// TwinCAT 3 PLC project DMXV2PLC
// ProgramVersion: 3.1.4023.0
// libraries:
//   Tc2_Math, * (Beckhoff Automation GmbH)
//   Tc2_Standard, * (Beckhoff Automation GmbH)
//   Tc2_System, * (Beckhoff Automation GmbH)
//   Tc2_Utilities, * (Beckhoff Automation GmbH)
//   Tc3_Module, * (Beckhoff Automation GmbH)
//   VisuDialogs, * (System)
//   VisuSymbols, * (System)
//   Base Interfaces,newest,System
// project tree:
//   DUTs/ arr_rt.TcDUT, ENUM_BufferMgmt.TcDUT (not stored), ENUM_IQ_OpMode.TcDUT, ENUM_I_ValRange.TcDUT, ENUM_I_Waveform.TcDUT (not stored), ENUM_SeqSM.TcDUT (not stored), ST_CSV_Record.TcDUT (not stored), typDMXInOut.TcDUT, typDMXInput.TcDUT, typDMXOutput.TcDUT, typFBDInOut.TcDUT, typFBDInput.TcDUT (not stored), typFBDOutput.TcDUT, typ_FBInt_Debounce.TcDUT (not stored), typ_FBInt_DMX.TcDUT (not stored)
//   / GlobalTextList.TcGTLO, PlcTask.TcTTO, Visualization Manager.TcVMO (not stored)
//   GVLs/ gc.TcGVL, gFB.TcGVL (not stored), GVL.TcGVL (not stored), g_ast.TcGVL
//   POUs/ DMXShop.TcPOU, DMXTest.TcPOU, FBOscillator.TcPOU, FB_DMX.TcPOU, FB_InputDebounce.TcPOU, f_to_Period.TcPOU (not stored), InterfaceLink.TcPOU, MAIN.TcPOU, Map.TcPOU (not stored), MapClamp.TcPOU (not stored), P_ArgToConvExample.TcPOU (not stored), P_BinaryModeRead.TcPOU (not stored), P_BinaryModeWrite.TcPOU (not stored), P_StringToConvExample.TcPOU (not stored), P_TextModeRead.TcPOU, P_TextModeWrite.TcPOU, SclByteDMX.TcPOU, SclBytePNP.TcPOU (not stored)
//   VISUs/ Visualization.TcVIS

CONFIGURATION DMXV2PLC
    RESOURCE PLC ON TwinCAT3
        TASK PlcTask(INTERVAL := T#10ms, PRIORITY := 20);
        PROGRAM InterfaceLink WITH PlcTask : InterfaceLink;
        PROGRAM P_TextModeRead WITH PlcTask : P_TextModeRead;
        PROGRAM DMXShop WITH PlcTask : DMXShop;
    END_RESOURCE
END_CONFIGURATION

// ---- DUTs/arr_rt.TcDUT
TYPE ARR_RT	 :
STRUCT
	arrRcvdR_T	: ARRAY[0..gc.uiMaxNrDMXTestCh] OF R_TRIG;
	arrExpctdBool : ARRAY[0..gc.uiMaxNrDMXTestCh] OF BOOL;
END_STRUCT
END_TYPE

// ---- DUTs/ENUM_IQ_OpMode.TcDUT
{attribute 'qualified_only'}
{attribute 'strict'}
TYPE ENUM_IQ_OpMode :
(
	EN_Cycle		:= 0,
	EN_LatchOn		:= 1,
	EN_OneShot		:= 2
);
END_TYPE

// ---- DUTs/ENUM_I_ValRange.TcDUT
{attribute 'qualified_only'}
{attribute 'strict'}
TYPE ENUM_I_ValRange :
(
	EN_8Bit		:= 0,
	EN_16Bit	:= 1
);
END_TYPE

// ---- DUTs/typDMXInOut.TcDUT
TYPE typDMXInOut :
STRUCT
	fOffset				: REAL; // 0-100% mapped to 8-bit (by Map Function)
	fLevel				: REAL; // 0-100% mapped to 8-bit (by Map Function)
	usiBitDepth			: USINT; // 1-8
	xCmdOn				: BOOL;
	xCmdOff				: BOOL;
	fOutputIncrement	: REAL;
	fFnGenerValTempSin	: LREAL;
	fFnGenerValRtn		: LREAL;
	uiMaxChannelVal		: UINT;
	uiMinChannelVal		: UINT;
	byMaxChanVal		: BYTE;
	byMinChanVal		: BYTE;
END_STRUCT
END_TYPE

// ---- DUTs/typDMXInput.TcDUT
TYPE typDMXInput :
STRUCT
	ENWaveform		: ENUM_I_Waveform;
	ENValRange		: ENUM_I_ValRange;
	fDutyCycle		: REAL; // just for Square Wave;
	fFrequency		: REAL;  // Frequency of cycling, expressed in Hz
	fOffset			: REAL; // 0-100% mapped to 8-bit (by Map Function)
	fLevel			: REAL; // 0-100% mapped to 8-bit (by Map Function)
	usiBitDepth		: USINT; // 1-8
	fPhase			: REAL; // 0-100% mapped to 8-bit (by Map Function)
	fDelay			: REAL; // 0-100% mapped to 8-bit (by Map Function)
	usiDelayDiv		: USINT; // to Delay the step of the Delay Divisor; for example, '2' would delay every second pulse by the amount spec'd by fDelay
	usiInputConfig	: USINT; // BYTE Value specified in USINT [0-255]
	xCmdOn				: BOOL;
	xCmdOff				: BOOL;
	fOutputIncrement	: REAL;
	fFnGenerValTempSin	: LREAL;
	fFnGenerValRtn		: LREAL;
	uiMaxChannelVal		: UINT;
	uiMinChannelVal		: UINT;
	byMaxChanVal		: BYTE;
	byMinChanVal		: BYTE;
END_STRUCT
END_TYPE

// ---- DUTs/typDMXOutput.TcDUT
TYPE typDMXOutput :
STRUCT
	byStatValue			: BYTE;
	fFnGeneratorVal		: REAL;
END_STRUCT
END_TYPE

// ---- DUTs/typFBDInOut.TcDUT
TYPE typFBDInOut :
	STRUCT
		xTrig		: BOOL;
	END_STRUCT
END_TYPE

// ---- DUTs/typFBDOutput.TcDUT
TYPE typFBDOutput :
STRUCT
	xGate	: BOOL;
END_STRUCT
END_TYPE

// ---- GVLs/gc.TcGVL
{attribute 'qualified_only'}
VAR_GLOBAL CONSTANT
	uiMaxNrOfDMXChannel				: UINT := 511;
	wChannelLength			AT %Q*	: WORD := 512;
	fPi								: REAL	:= 3.141592653589793238462643383279;
	uiMinNrDMXTestCh				: UINT	:= 0;
	uiMaxNrDMXTestCh				: UINT	:= 79; // Dictated by hardware constraints (80 channels input)
	uiChannelsUT	 				: UINT	:= 80;		(*Channels Under Test *)
	uiVisualizationIndexLim			: UINT	:= 7;
	uiDUTConfigCountSplit			: UINT	:= 255;
	uiChannelSplitCount				: UINT	:= 256;
	
	// DMXShop 
	RED		: USINT := 0;
	GREEN 	: USINT := 1;
	BLUE	: USINT := 2;
	WHITE	: USINT := 3;

END_VAR

// ---- GVLs/g_ast.TcGVL
{attribute 'qualified_only'}
VAR_GLOBAL
		// INPUT array structs for mapping to Physical I/O (PIO)
//	gast_SensorInput		AT %I* : ARRAY[0..gc.usiMaxNrOfSensor] OF typ_FBInt_Debounce;
	
	//2 Sensors on each valve (assumed)
//	gast_ValveSensorInput	AT %I* : ARRAY[0..(2*gc.usiMaxNrOfValveCtrl)] OF typ_FBInt_Debounce;
//	gast_AnalogInput		AT %I* : ARRAY[0..gc.usiMaxNrOfAnalogIn] OF typ_FBInt_Analog;
	
// OUTPUT array structs for mapping to Physical I/O (PIO)
//	gast_ValveCtrlOutput	AT %Q* : ARRAY[0..gc.usiMaxNrOfValveCtrl] OF typ_FBInt_ValveCtrl;
//	gast_DigCtrlOutput		AT %Q* : ARRAY[0..gc.usiMaxNrOfDigCtrl] OF typ_FBInt_DigCtrl;
	DMX						: ARRAY[0..gc.uiMaxNrOfDMXChannel] OF typ_FBInt_DMX;
	DMXPhysOut				: ARRAY[0..gc.uiMaxNrOfDMXChannel] OF BYTE; (* software buffer *)
	DMXHWOut		AT %Q*	: ARRAY[0..gc.uiMaxNrOfDMXChannel] OF BYTE; (* Defined to allow Multi-Link of I/O in Physical I/O tree *)
	arrFBIntPNP				: ARRAY[0..gc.uiMaxNrDMXTestCh] OF typ_FBInt_Debounce;
	arrFBIntNPN				: ARRAY[0..gc.uiMaxNrDMXTestCh] OF typ_FBInt_Debounce;
	arrInputPNP		AT %I*	: ARRAY[0..gc.uiMaxNrDMXTestCh] OF BOOL;
	arrInputNPN		AT %I*	: ARRAY[0..gc.uiMaxNrDMXTestCh] OF BOOL;
END_VAR

// ---- POUs/InterfaceLink.TcPOU
PROGRAM InterfaceLink
VAR
	iResult					: INT;
	iLoopFBAnalogIn			: INT;
	iLoopFBSensor			: INT;
	iLoopFBValveSensor		: INT;
	iLoopFBDigCtrl			: INT;
	iLoopFBValveCtrl		: INT;
	uiLoopDMXCtrlI			: UINT;
	uiLoopDMXCtrlII			: UINT;
	uiLoopDebouncePNPI		: UINT;
	uiLoopDebounceNPNI		: UINT;
	uiForLoopDMXI10			: UINT;
	uiForLoopDMXI11			: UINT;
	uiForLoopDMXI12			: UINT;
	uiForLoopDebouncePNP	: UINT;
	uiForLoopDebounceNPN	: UINT;
END_VAR

//Call all the I/O Function Blocks continuously; link to array-structs with every call;
(*
FOR iLoopFBAnalogIn := 0 TO gc.usiMaxNrOfAnalogIn BY 1 DO
	gFB.arrFB_AnalogInput[iLoopFBAnalogIn](I:=gast_AnalogInput[iLoopFBAnalogIn].I, IQ:=gast_AnalogInput[iLoopFBAnalogIn].IQ, Q=>gast_AnalogInput[iLoopFBAnalogIn].Q);
END_FOR

FOR iLoopFBSensor := 0 TO gc.usiMaxNrOfSensor BY 1 DO
	gFB.arrFB_Sensor[iLoopFBSensor](I:=gast_SensorInput[iLoopFBSensor].I, IQ:=gast_SensorInput[iLoopFBSensor].IQ, Q=>gast_SensorInput[iLoopFBSensor].Q);
END_FOR

FOR iLoopFBValveSensor := 0 TO (2*gc.usiMaxNrOfValveCtrl) BY 1 DO
	gFB.arrFB_Sensor[iLoopFBValveSensor](I:=gast_ValveSensorInput[iLoopFBValveSensor].I, IQ:=gast_ValveSensorInput[iLoopFBValveSensor].IQ, Q=>gast_ValveSensorInput[iLoopFBValveSensor].Q);
END_FOR

FOR iLoopFBDigCtrl := 0 TO gc.usiMaxNrOfSensor BY 1 DO
	gFB.arrFB_DigCtrl[iLoopFBDigCtrl](I:=gast_DigCtrlOutput[iLoopFBDigCtrl].I, IQ:=gast_DigCtrlOutput[iLoopFBDigCtrl].IQ, Q=>gast_DigCtrlOutput[iLoopFBDigCtrl].Q);
END_FOR

FOR iLoopFBValveCtrl := 0 TO gc.usiMaxNrOfValveCtrl BY 1 DO
	gFB.arrFB_ValveCtrl[iLoopFBValveCtrl](I:=gast_ValveCtrlOutput[iLoopFBValveCtrl].I, IQ:=gast_ValveCtrlOutput[iLoopFBValveCtrl].IQ, Q=>gast_ValveCtrlOutput[iLoopFBValveCtrl].Q);
END_FOR
*)
FOR uiLoopDMXCtrlI := 0 TO gc.uiMaxNrOfDMXChannel BY 1 DO
	gFB.arrFB_DMX[uiLoopDMXCtrlI]();
END_FOR

//Expose an array of bytes that can be ultimately 'multi-linked' to hardware
FOR uiLoopDMXCtrlII := 0 TO gc.uiMaxNrOfDMXChannel BY 1 DO
	g_ast.DMXPhysOut[uiLoopDMXCtrlII]	:= gFB.arrFB_DMX[uiLoopDMXCtrlII].Q.byStatValue;
END_FOR

//Debounce PNP
FOR uiLoopDebouncePNPI	:= 0 TO gc.uiMaxNrDMXTestCh BY 1 DO
	gFB.arrFB_DebouncePNP[uiLoopDebouncePNPI](I:=g_ast.arrFBIntPNP[uiLoopDebouncePNPI].I, IQ:=g_ast.arrFBIntPNP[uiLoopDebouncePNPI].IQ, Q=>g_ast.arrFBIntPNP[uiLoopDebouncePNPI].Q);
END_FOR

//Debounce NPN
FOR uiLoopDebounceNPNI	:= 0 TO gc.uiMaxNrDMXTestCh BY 1 DO
	gFB.arrFB_DebounceNPN[uiLoopDebounceNPNI](I:=g_ast.arrFBIntNPN[uiLoopDebounceNPNI].I, IQ:=g_ast.arrFBIntNPN[uiLoopDebounceNPNI].IQ, Q=>g_ast.arrFBIntNPN[uiLoopDebounceNPNI].Q);
END_FOR

//Link all the user-specified params to the respective Function Blocks
//RED

(*
RGB PARAMETERS - Hence, the Groups of 4 incremented in this way;

FOR iForLoopDMXI1:= 0 TO gc.uiMaxNrOfDMXChannel BY 4 DO
	g_ast.DMX[iForLoopDMXI1].I.ENWaveform		:= ENUM_I_Waveform.EN_Sin; //"50% duty cycle"
	g_ast.DMX[iForLoopDMXI1].I.fDutyCycle		:= 50; // %
	g_ast.DMX[iForLoopDMXI1].I.fLevel			:= iSlider5; //%
	g_ast.DMX[iForLoopDMXI1].I.fOffset			:= 0; // %
	g_ast.DMX[iForLoopDMXI1].I.usiBitDepth		:= 8; // 0-8, or 0-16, depending
	g_ast.DMX[iForLoopDMXI1].I.fPhase			:= 0; // %
	g_ast.DMX[iForLoopDMXI1].I.fDelay			:= 0; // %
	g_ast.DMX[iForLoopDMXI1].I.usiDelayDiv		:= 0; // which step to have delay applied
END_FOR

//GREEN
FOR iForLoopDMXI2:= 1 TO gc.uiMaxNrOfDMXChannel BY 4 DO
	g_ast.DMX[iForLoopDMXI2].I.ENWaveform		:= ENUM_I_Waveform.EN_Sin; //"50% duty cycle"
	g_ast.DMX[iForLoopDMXI2].I.fDutyCycle		:= 50; // %
	g_ast.DMX[iForLoopDMXI2].I.fLevel			:= iSlider6; //%
	g_ast.DMX[iForLoopDMXI2].I.fOffset			:= 0; // %
	g_ast.DMX[iForLoopDMXI2].I.usiBitDepth		:= 8; // 0-8, or 0-16, depending
	g_ast.DMX[iForLoopDMXI2].I.fPhase			:= 0; // %
	g_ast.DMX[iForLoopDMXI2].I.fDelay			:= 0; // %
	g_ast.DMX[iForLoopDMXI2].I.usiDelayDiv		:= 0; // which step to have delay applied
END_FOR

//BLUE
FOR iForLoopDMXI3:= 2 TO gc.uiMaxNrOfDMXChannel BY 4 DO
	g_ast.DMX[iForLoopDMXI3].I.ENWaveform		:= ENUM_I_Waveform.EN_Sin; //"50% duty cycle"
	g_ast.DMX[iForLoopDMXI3].I.fDutyCycle		:= 50; // %
	g_ast.DMX[iForLoopDMXI3].I.fLevel			:= iSlider7; //%
	g_ast.DMX[iForLoopDMXI3].I.fOffset			:= 0; // %
	g_ast.DMX[iForLoopDMXI3].I.usiBitDepth		:= 8; // 0-8, or 0-16, depending
	g_ast.DMX[iForLoopDMXI3].I.fPhase			:= 0; // %
	g_ast.DMX[iForLoopDMXI3].I.fDelay			:= 0; // %
	g_ast.DMX[iForLoopDMXI3].I.usiDelayDiv		:= 0; // which step to have delay applied
END_FOR

//WHITE
FOR iForLoopDMXI4:= 3 TO gc.uiMaxNrOfDMXChannel BY 4 DO
	g_ast.DMX[iForLoopDMXI4].I.ENWaveform		:= ENUM_I_Waveform.EN_Sin; //"50% duty cycle"
	g_ast.DMX[iForLoopDMXI4].I.fDutyCycle		:= 50; // %
	g_ast.DMX[iForLoopDMXI4].I.fLevel			:= iSlider8; //%
	g_ast.DMX[iForLoopDMXI4].I.fOffset			:= 0; // %
	g_ast.DMX[iForLoopDMXI4].I.usiBitDepth		:= 8; // 0-8, or 0-16, depending
	g_ast.DMX[iForLoopDMXI4].I.fPhase			:= 0; // %
	g_ast.DMX[iForLoopDMXI4].I.fDelay			:= 0; // %
	g_ast.DMX[iForLoopDMXI4].I.usiDelayDiv		:= 0; // which step to have delay applied
END_FOR


FOR iForLoopDMXI5	:= 0 TO gc.uiMaxNrOfDMXChannel BY 4 DO 
	g_ast.DMX[iForLoopDMXI5].I.fFrequency		:= iSlider1; //Hz
END_FOR

FOR iForLoopDMXI6	:= 0 TO gc.uiMaxNrOfDMXChannel BY 4 DO 
	g_ast.DMX[iForLoopDMXI6].I.fFrequency		:= iSlider2; //Hz
END_FOR

FOR iForLoopDMXI7	:= 0 TO gc.uiMaxNrOfDMXChannel BY 4 DO 
	g_ast.DMX[iForLoopDMXI7].I.fFrequency		:= iSlider3; //Hz
END_FOR

FOR iForLoopDMXI8	:= 0 TO gc.uiMaxNrOfDMXChannel BY 4 DO 
	g_ast.DMX[iForLoopDMXI8].I.fFrequency		:= iSlider4; //Hz
END_FOR
*)

FOR uiForLoopDMXI10:= 0 TO gc.uiDUTConfigCountSplit BY 1 DO
	gFB.arrFB_DMX[uiForLoopDMXI10].I.fFrequency		:= 0;
	gFB.arrFB_DMX[uiForLoopDMXI10].I.ENWaveform		:= ENUM_I_Waveform.EN_GateCtrl;
	gFB.arrFB_DMX[uiForLoopDMXI10].I.ENValRange		:= ENUM_I_ValRange.EN_8Bit;
	gFB.arrFB_DMX[uiForLoopDMXI10].I.fDutyCycle		:= 100; // %
	gFB.arrFB_DMX[uiForLoopDMXI10].I.fLevel			:= 100; //%
	gFB.arrFB_DMX[uiForLoopDMXI10].I.fOffset		:= 0; // %
	gFB.arrFB_DMX[uiForLoopDMXI10].I.usiBitDepth	:= 8; // 0-8, or 0-16, depending
	gFB.arrFB_DMX[uiForLoopDMXI10].I.fPhase			:= 0; // %
	gFB.arrFB_DMX[uiForLoopDMXI10].I.fDelay			:= 0; // %
	gFB.arrFB_DMX[uiForLoopDMXI10].I.usiDelayDiv	:= 0; // which step to have delay applied
//	g_ast.DMX[uiForLoopDMXI10].I.fFrequency		:= 0;
//	g_ast.DMX[uiForLoopDMXI10].I.ENWaveform		:= ENUM_I_Waveform.EN_GateCtrl;
//	g_ast.DMX[uiForLoopDMXI10].I.ENValRange		:= ENUM_I_ValRange.EN_8Bit;
//	g_ast.DMX[uiForLoopDMXI10].I.fDutyCycle		:= 100; // %
//	g_ast.DMX[uiForLoopDMXI10].I.fLevel			:= 100; //%
//	g_ast.DMX[uiForLoopDMXI10].I.fOffset		:= 0; // %
//	g_ast.DMX[uiForLoopDMXI10].I.usiBitDepth	:= 8; // 0-8, or 0-16, depending
//	g_ast.DMX[uiForLoopDMXI10].I.fPhase			:= 0; // %
//	g_ast.DMX[uiForLoopDMXI10].I.fDelay			:= 0; // %
//	g_ast.DMX[uiForLoopDMXI10].I.usiDelayDiv	:= 0; // which step to have delay applied
//Channels for Configuration of testing on other DMX Channels;
END_FOR

FOR uiForLoopDMXI11:= gc.uiChannelSplitCount TO gc.uiMaxNrOfDMXChannel BY 1 DO
	gFB.arrFB_DMX[uiForLoopDMXI11].I.fFrequency		:= 0;
	gFB.arrFB_DMX[uiForLoopDMXI11].I.ENWaveform		:= ENUM_I_Waveform.EN_GateConfig;
	gFB.arrFB_DMX[uiForLoopDMXI11].I.ENValRange		:= ENUM_I_ValRange.EN_8Bit;
	gFB.arrFB_DMX[uiForLoopDMXI11].I.fDutyCycle		:= 100; // %
	gFB.arrFB_DMX[uiForLoopDMXI11].I.fLevel			:= 100; //%
	gFB.arrFB_DMX[uiForLoopDMXI11].I.fOffset		:= 0; // %
	gFB.arrFB_DMX[uiForLoopDMXI11].I.usiBitDepth	:= 8; // 0-8, or 0-16, depending
	gFB.arrFB_DMX[uiForLoopDMXI11].I.fPhase			:= 0; // %
	gFB.arrFB_DMX[uiForLoopDMXI11].I.fDelay			:= 0; // %
	gFB.arrFB_DMX[uiForLoopDMXI11].I.usiDelayDiv	:= 0; // which step to have delay applied
//	g_ast.DMX[uiForLoopDMXI10].I.fFrequency		:= 0;
//	g_ast.DMX[uiForLoopDMXI10].I.ENWaveform		:= ENUM_I_Waveform.EN_GateConfig;
//	g_ast.DMX[uiForLoopDMXI10].I.ENValRange		:= ENUM_I_ValRange.EN_8Bit;
//	g_ast.DMX[uiForLoopDMXI10].I.fDutyCycle		:= 100; // %
//	g_ast.DMX[uiForLoopDMXI10].I.fLevel			:= 100; //%
//	g_ast.DMX[uiForLoopDMXI10].I.fOffset		:= 0; // %
//	g_ast.DMX[uiForLoopDMXI10].I.usiBitDepth	:= 8; // 0-8, or 0-16, depending
//	g_ast.DMX[uiForLoopDMXI10].I.fPhase			:= 0; // %
//	g_ast.DMX[uiForLoopDMXI10].I.fDelay			:= 0; // %
//	g_ast.DMX[uiForLoopDMXI10].I.usiDelayDiv	:= 0; // which step to have delay applied
//Channels for Configuration of testing on other DMX Channels;
END_FOR

//Input Debounce Params PNP
FOR uiForLoopDebouncePNP	:= 0 TO gc.uiMaxNrDMXTestCh BY 1 DO
	g_ast.arrFBIntPNP[uiForLoopDebouncePNP].I.tOnDelay	:= T#0S;
	g_ast.arrFBIntPNP[uiForLoopDebouncePNP].I.tOffDelay	:= T#10MS;
END_FOR

//Input Debounce Params NPN
FOR uiForLoopDebounceNPN	:= 0 TO gc.uiMaxNrDMXTestCh BY 1 DO
	g_ast.arrFBIntNPN[uiForLoopDebounceNPN].I.tOnDelay	:= T#0S;
	g_ast.arrFBIntNPN[uiForLoopDebounceNPN].I.tOffDelay	:= T#3MS;
END_FOR

//Read the CSV Parameters into the DMX FBs - via the "mediating" Config arrays
FOR uiForLoopDMXI12:= 0 TO gc.uiMaxNrOfDMXChannel BY 1 DO
	gFB.arrFB_DMX[uiForLoopDMXI12].I.usiInputConfig	:= 	DMXTest.arr_usiRecipeSetting[uiForLoopDMXI12];
END_FOR

END_PROGRAM

// ---- POUs/DMXTest.TcPOU
PROGRAM DMXTest
VAR
	xConfigSet					: BOOL;
	xStatTestInProgress			: BOOL;
	xDMXSeqTestInProgressOnce	: BOOL;
	xDMXSeqTestInProgressTwice	: BOOL;
	xDMXSeqTestInProgressOnceDC	: BOOL;
	uiCounter2					: UINT;
	uiCounter3					: UINT;
	uiCounter4					: UINT;
	uiCounter5					: UINT;
	uiCounter6					: UINT;
	uiCounter7					: UINT;
	uiCounter8					: UINT;
	uiCounter9					: UINT;
	uiDedicatedRcvdRTIndex		: UINT;
	uiContinuousRTIndex			: UINT;
	
	uiForLoopCfgIndex			: UINT;
//	uiForLoopCtrlWriteIndex		: UINT;
//	uiForLoopCtrlWriteIndex2	: UINT;	
	uiLoopExpctdIndex			: UINT;
	uiForLoopClearExpctd		: UINT;
	uiLoopRcvIndex				: UINT;
	uiByteIndex					: UINT;
	iForLoopRecipeFindMin		: INT;
	iForLoopRecipeFindMax		: INT;
	iForLoopRecipeFindMax1		: INT;
	iForLoopRecipeMin			: INT;
	uiForLoopRecipe				: UINT;
	uiLoopIterDMXDUTArraySeq	: UINT;
	uiLoopIterDMXDUTArrayM		: UINT;
	uiLoopIterDUTArray24V		: UINT;
	uiLoopIterDUTArrayGND		: UINT;
	uiLoopIterTestArrSeq		: UINT;
	uiLoopIterTestArrM			: UINT;
	uiLoopIterTestArr24V		: UINT;
	uiLoopIterTestArrGND		: UINT;	
	iCompareStaticSM			: INT;
	iCompareSeq					: ARRAY[0..ENUM_SeqSM.Twice] OF INT;
	iParseFile					: INT;
	iSetConfig					: INT;
	iSetExpctdBufferSM			: INT;
	iReindexExpctedBufferSM		: INT;
	rt_RunStaticTest			: R_TRIG;
	rt_RunSeqTestOnce			: R_TRIG;
	rt_RunSeqTestOnceDC			: R_TRIG;
	rt_RunSeqTestTwice			: R_TRIG;
	rt_ResetTest				: R_TRIG;
	rt_ResetTestSeq				: R_TRIG;
	rt_ResetTestSeqDC			: R_TRIG;
	r_tStaticTestDone			: R_TRIG;
	
	//Arrays (Refactor 30-09-21)
	arr_uiRecipeIndexTmp		: ARRAY[0..gc.uiDUTConfigCountSplit] OF UINT;
 	arruiDMXChDUTTmp			: ARRAY[0..gc.uiDUTConfigCountSplit] OF UINT;
	arrsDUTChTypeTmp			: ARRAY[0..gc.uiDUTConfigCountSplit] OF STRING[3];	
	arr_uiRecipeIndex			: ARRAY[0..gc.uiDUTConfigCountSplit] OF UINT;
 	arruiDMXChDUT				: ARRAY[0..gc.uiDUTConfigCountSplit] OF UINT;
	arrsDUTChType				: ARRAY[0..gc.uiDUTConfigCountSplit] OF STRING[3];
	xFileImported				: BOOL;
	arr_usiRecipeSettingTmp		: ARRAY[0..gc.uiMaxNrOfDMXChannel] OF USINT;
	arr_usiRecipeSetting		: ARRAY[0..gc.uiMaxNrOfDMXChannel] OF USINT;






	
		
	arrxRcvdBufferPNP24V		: ARRAY[0..gc.uiMaxNrDMXTestCh] OF BOOL;
	arrxRcvdBufferNPN24V		: ARRAY[0..gc.uiMaxNrDMXTestCh] OF BOOL;
	arrxRcvdBufferPNPGND		: ARRAY[0..gc.uiMaxNrDMXTestCh] OF BOOL;
	arrxRcvdBufferNPNGND		: ARRAY[0..gc.uiMaxNrDMXTestCh] OF BOOL;
	
	arrxRcvdBufferPNPSeq		: ARRAY[0..gc.uiMaxNrDMXTestCh] OF BOOL;
	arrxRcvdBufferNPNSeq		: ARRAY[0..gc.uiMaxNrDMXTestCh] OF BOOL;	
	arrxRcvdBufferPNPMotor		: ARRAY[0..gc.uiMaxNrDMXTestCh] OF BOOL;
	arrxRcvdBufferNPNMotor		: ARRAY[0..gc.uiMaxNrDMXTestCh] OF BOOL;
	
	arrxExpctdPNP				: ARRAY[0..gc.uiMaxNrOfDMXChannel] OF BOOL; //What is expected based on the recipe file
	arrxExpctdNPN				: ARRAY[0..gc.uiMaxNrOfDMXChannel] OF BOOL; //What is expected based on the recipe file
	arrxExpctdTmpPNP			: ARRAY[0..gc.uiMaxNrOfDMXChannel] OF BOOL; //What is expected based on the recipe file, reindexed from DUT (usually 0)
	arrxExpctdTmpNPN			: ARRAY[0..gc.uiMaxNrOfDMXChannel] OF BOOL; //What is expected based on the recipe file, reindexed from DUT (usually 0)
	arrxExpctdTmpPNP24V			: ARRAY[0..gc.uiMaxNrDMXTestCh] OF BOOL; //What is expected based on the recipe file, reindexed from DUT (usually 0)
	arrxExpctdTmpNPN24V			: ARRAY[0..gc.uiMaxNrDMXTestCh] OF BOOL; //What is expected based on the recipe file, reindexed from DUT (usually 0)
	arrxExpctdTmpPNPGND			: ARRAY[0..gc.uiMaxNrDMXTestCh] OF BOOL; //What is expected based on the recipe file, reindexed from DUT (usually 0)
	arrxExpctdTmpNPNGND			: ARRAY[0..gc.uiMaxNrDMXTestCh] OF BOOL; //What is expected based on the recipe file, reindexed from DUT (usually 0)

	arrxExpctdTmpPNPSeqDMX		: ARRAY[0..gc.uiMaxNrDMXTestCh] OF BOOL; //What is expected based on the recipe file, reindexed from DUT (usually 0)
	arrxExpctdTmpNPNSeqDMX		: ARRAY[0..gc.uiMaxNrDMXTestCh] OF BOOL; //What is expected based on the recipe file, reindexed from DUT (usually 0)
	arrxExpctdTmpPNPSeqDC		: ARRAY[0..gc.uiMaxNrDMXTestCh] OF BOOL; //What is expected based on the recipe file, reindexed from DUT (usually 0)
	arrxExpctdTmpNPNSeqDC		: ARRAY[0..gc.uiMaxNrDMXTestCh] OF BOOL; //What is expected based on the recipe file, reindexed from DUT (usually 0)

	arrxExpctdTmpPNPSeq			: ARRAY[0..gc.uiMaxNrOfDMXChannel] OF BOOL; //What is expected based on the recipe file, reindexed from DUT (usually 0)
	arrxExpctdTmpNPNSeq			: ARRAY[0..gc.uiMaxNrOfDMXChannel] OF BOOL; //What is expected based on the recipe file, reindexed from DUT (usually 0)
	arrxExpctdTmpPNPMotor		: ARRAY[0..gc.uiMaxNrOfDMXChannel] OF BOOL; //What is expected based on the recipe file, reindexed from DUT (usually 0)
	arrxExpctdTmpNPNMotor		: ARRAY[0..gc.uiMaxNrOfDMXChannel] OF BOOL; //What is expected based on the recipe file, reindexed from DUT (usually 0)
	
	arrxExpctdMaskPNPSeq		: ARRAY[0..gc.uiMaxNrOfDMXChannel] OF BOOL; //Copy the contents of hardware buffer 
	arrxExpctdMaskNPNSeq		: ARRAY[0..gc.uiMaxNrOfDMXChannel] OF BOOL; //Copy the contents of hardware buffer 
	arr_diTestStaticPNP24V		: ARRAY[0..gc.uiMaxNrDMXTestCh] OF DINT;
	arr_diTestStaticNPN24V		: ARRAY[0..gc.uiMaxNrDMXTestCh] OF DINT;
	arr_diTestStaticPNPGND		: ARRAY[0..gc.uiMaxNrDMXTestCh] OF DINT;
	arr_diTestStaticNPNGND		: ARRAY[0..gc.uiMaxNrDMXTestCh] OF DINT;
	arr_diTestPNPSeqOnceLine			: ARRAY[0..gc.uiMaxNrDMXTestCh] OF DINT;
	arr_diTestPNPSeqOnceLineTmp			: ARRAY[0..gc.uiMaxNrDMXTestCh] OF DINT;
	arr_diTestNPNSeqOnceLine			: ARRAY[0..gc.uiMaxNrDMXTestCh] OF DINT;
	arr_diTestNPNSeqOnceLineTmp			: ARRAY[0..gc.uiMaxNrDMXTestCh] OF DINT;

	arr_udiMEMCPYPNPSeqOnceRcvdTmp		: ARRAY[0..gc.uiMaxNrDMXTestCh] OF UDINT;
	arr_udiMEMCPYNPNSeqOnceRcvdTmp		: ARRAY[0..gc.uiMaxNrDMXTestCh] OF UDINT;
			
	diTestStaticPNP24V				: DINT;
	diTestStaticNPN24V				: DINT;
	diTestStaticPNPGND				: DINT;	
	diTestStaticNPNGND				: DINT;
	
	diTestPNPSeqOnceComplete		: DINT;

	arrdiTestPNPSeqOnceComplete		: ARRAY[0..gc.uiMaxNrDMXTestCh] OF DINT;
	arrdiTestPNPSeqOnceCompleteTmp	: ARRAY[0..gc.uiMaxNrDMXTestCh] OF DINT;

	arrdiTestNPNSeqOnceComplete		: ARRAY[0..gc.uiMaxNrDMXTestCh] OF DINT;
	arrdiTestNPNSeqOnceCompleteTmp	: ARRAY[0..gc.uiMaxNrDMXTestCh] OF DINT;

	arrdiTestNPNSeqOnceCompleteProblemIndex		: ARRAY[0..gc.uiMaxNrDMXTestCh] OF DINT;
	
	arrudiStaticCopyResultPNP24V	: ARRAY[0..gc.uiMaxNrOfDMXChannel] OF UDINT;
	arrudiStaticCopyResultNPN24V	: ARRAY[0..gc.uiMaxNrOfDMXChannel] OF UDINT;
	arrudiStaticCopyResultPNPGND	: ARRAY[0..gc.uiMaxNrOfDMXChannel] OF UDINT;
	arrudiStaticCopyResultNPNGND	: ARRAY[0..gc.uiMaxNrOfDMXChannel] OF UDINT;	

	arr_diTestPNPMotorDir1		: ARRAY[0..gc.uiMaxNrDMXTestCh] OF DINT;
	arr_diTestNPNMotorDir1		: ARRAY[0..gc.uiMaxNrDMXTestCh] OF DINT;
	arr_diTestPNPMotorDir2		: ARRAY[0..gc.uiMaxNrDMXTestCh] OF DINT;
	arr_diTestNPNMotorDir2		: ARRAY[0..gc.uiMaxNrDMXTestCh] OF DINT;

	
	
	diCompTestResult			: DINT;
	diCompTestResultTemp		: DINT;
	diTestResultStaticPNP		: DINT;
	diTestResultStaticNPN		: DINT;	

	arrVisu_diTestResult		: ARRAY[0..gc.uiMaxNrDMXTestCh] OF DINT;
	uiVisuIndex					: UINT;
	tonReadWait					: TON;
	tonConvert					: TON;
	tonWriteCopyWait			: TON;
	tonTestIterGap				: TON;
	tTestTime					: TIME;
	tWriteWaitTime				: TIME;
	r_tSetConfig				: R_TRIG;
	uiRecipeIndexRcv			: UINT;
	uiMinRecipeIndex			: UINT;
	uiMaxRecipeIndex			: UINT;
	cuiMinDUTIndex				: UINT	:= 0; // Constant
	uiMaxRecipeIndexTemp		: UINT;
	arruiMotorTestIndices		: ARRAY[0..gc.uiMaxNrOfDMXChannel] OF UINT;
	arruiMotorTestIndicesTmp	: ARRAY[0..gc.uiMaxNrOfDMXChannel] OF UINT;
	arruiSeqTestIndices			: ARRAY[0..gc.uiMaxNrOfDMXChannel] OF UINT;
	arruiSeqTestIndicesTmp		: ARRAY[0..gc.uiMaxNrOfDMXChannel] OF UINT;
	
	arruiSeqTestIndicesDMX			: ARRAY[0..gc.uiMaxNrDMXTestCh] OF UINT;
	arruiSeqTestIndicesDMXSW		: ARRAY[0..gc.uiMaxNrDMXTestCh] OF UINT;
	arruiSeqTestIndicesDMXTmp		: ARRAY[0..gc.uiMaxNrDMXTestCh] OF UINT;
	
	arruiSeqTestIndicesDC			: ARRAY[0..gc.uiMaxNrDMXTestCh] OF UINT;
	arruiSeqTestIndicesDCTmp		: ARRAY[0..gc.uiMaxNrDMXTestCh] OF UINT;	
	
	arrui24VTestIndices			: ARRAY[0..gc.uiMaxNrOfDMXChannel] OF UINT;
	arrui24VTestIndicesTmp		: ARRAY[0..gc.uiMaxNrOfDMXChannel] OF UINT;
	arruiGNDTestIndices			: ARRAY[0..gc.uiMaxNrOfDMXChannel] OF UINT;
	arruiGNDTestIndicesTmp		: ARRAY[0..gc.uiMaxNrOfDMXChannel] OF UINT;
	udiMemCpyResultPNP			: UDINT;
	udiMemCpyResultDMX			: UDINT;	
	r_tSetExpectedBuff			: R_TRIG;
	r_tExpectedBufferSet		: R_TRIG;
	uiLoopExpctdIndexRead		: UINT;
	uiLoopExpctdIndexWrite		: UINT;
	xTestBoolDelete				: BOOL;
	uiForLoopZeroStorageArray	: UINT;
	
	//For DUT Config
	r_tSetDUTVal				: R_TRIG;
	usiDUTVal					: USINT;
	uiForLoopDUTIter			: UINT;
	iSetDUTSM					: INT;
	
	//For 'Invert Recipe Settings'
	uiStartingIndex				: UINT;
	uiEndingIndex				: UINT;
	uiRecipeInvertIter			: UINT;
	R_TInvertRecipe				: R_TRIG;
	iInvertRecipeSM				: INT;
END_VAR

SeqTestOnce();
//SeqTestTwice();
//SeqTestOnceDC();
InvertRecipeSettings();
rt_RunStaticTest();
rt_ResetTest();
r_tSetConfig();//Set config when file is loaded; this condition happens when End-of-File (EOF) is reached; set by HMI button
r_tSetExpectedBuff(CLK:=r_tSetConfig.Q);
r_tExpectedBufferSet();
r_tStaticTestDone(CLK			:= (iCompareStaticSM = 110));
r_tSetDUTVal();
tonReadWait(PT		:= tTestTime);
tonConvert(PT		:= tTestTime);
tonWriteCopyWait(PT	:= tWriteWaitTime);
tonTestIterGap(PT	:= tTestTime);
tTestTime			:= T#80MS;
//just an example one
tWriteWaitTime		:= T#10MS; // same as the tOffDelay set to the input debounce FB
//DMX DUT Channels, Software 0-255 
//DMX Config Channels, Software, 256-511
//DMX DUT Channels, Hardware 1-256
//DMX Config Channels, Hardware, 257-512

//Interface Link - continued - DMXTest Local Vars

//"Config Complete" Expctd Buffer, and "Config Complete" Received Buffer; then Global Comparison is like 'masking' all but one channel at a time;

CASE iParseFile OF

0:
IF P_TextModeRead.r_tFileChg.Q THEN
	xFileImported		:= FALSE;	
	iParseFile			:= 5;
END_IF

5:
IF P_TextModeRead.fbFileGets.bEOF THEN
	uiForLoopRecipe	:= 0; // Reset the iterator used in the next state of the SM
	iParseFile		:= 10;
END_IF
	
10://At first check for any recipe items specified in the file;
//Load the recipe data into respective arrays
//For recipe indices = 0 to 255, parse the file to read the recipe index, DMX channel, and channel type
FOR uiForLoopRecipe := 0 TO gc.uiDUTConfigCountSplit BY 1 DO
	//Read the Recipe Index
	arr_uiRecipeIndexTmp[uiForLoopRecipe]		:= STRING_TO_UINT(P_TextModeRead.database[uiForLoopRecipe,0]);
	//Read the DMX Channel for the DUT
	arruiDMXChDUTTmp[uiForLoopRecipe]			:= STRING_TO_UINT(P_TextModeRead.database[uiForLoopRecipe,1]);
	//Read the type of Channel on the DUT
	arrsDUTChTypeTmp[uiForLoopRecipe]			:= P_TextModeRead.database[uiForLoopRecipe,2];
END_FOR
//Stash the values from temp (inside FOR loop) to other arrays
arr_uiRecipeIndex	:= arr_uiRecipeIndexTmp;
arruiDMXChDUT		:= arruiDMXChDUTTmp;
arrsDUTChType		:= arrsDUTChTypeTmp;

//If the 'TextModeRead' re-enters 'Ready' state then advance this SM
IF P_TextModeRead.step = 0 THEN
	xFileImported		:= TRUE;
	iParseFile			:= 0;	
END_IF

END_CASE

CASE iSetConfig OF

//Don't look at the P_TextRead; evaluate on the arrays you just imported

0:
IF r_tSetConfig.Q THEN
	iSetConfig			:= 10;	
END_IF

10://Read the string that is loaded from file reader; pass value to DMX Function Block, at the appropriate Config index
//This is the setting to control the position of the 'config' relays on the tester
//Ensure that the declared arrays are sufficiently long to handle the max conceivable value (512 x 2, in this case?)
FOR uiForLoopRecipe := 0 TO gc.uiDUTConfigCountSplit BY 1 DO
	IF (arruiDMXChDUT[uiForLoopRecipe] <> 0) THEN
		//Set the config routing := NPN
		arr_usiRecipeSettingTmp[(uiForLoopRecipe+gc.uiChannelSplitCount)]	:= 255;
	ELSIF (arruiDMXChDUT[uiForLoopRecipe] = 0) THEN
		//Set the config routing := PNP
		arr_usiRecipeSettingTmp[(uiForLoopRecipe+gc.uiChannelSplitCount)]	:= 0;
	END_IF	
END_FOR
//Stash the values from temp (inside FOR loop) to other arrays
arr_usiRecipeSetting	:= arr_usiRecipeSettingTmp;

	iSetConfig			:= 20;	

20://Iterate over the config listings to create indices for what must be tested static (power, ground), and what must be tested sequentially (channels)
uiLoopIterDMXDUTArraySeq	:= 0;
uiLoopIterTestArrSeq		:= 0;
//Zero out the array that is copied to in the next state of the SM
FOR uiForLoopZeroStorageArray	:= 0 TO gc.uiMaxNrOfDMXChannel BY 1 DO
	arruiSeqTestIndicesTmp[uiForLoopZeroStorageArray]	:= 0;
END_FOR
//Stash the values from temp (inside FOR loop) to other arrays
arruiSeqTestIndices		:= arruiSeqTestIndicesTmp;
iSetConfig				:= 40;	

40:
//For any 'DMX'-type channels with an assigned channel # (from the recipe), then copy only those elements to another array
//These are elements that are tested sequentially - once - so this includes Dry Contacts but not Motors
REPEAT
	IF ((arrsDUTChType[uiLoopIterDMXDUTArraySeq] = 'DMX') OR (arrsDUTChType[uiLoopIterDMXDUTArraySeq] = '24V')) AND (arruiDMXChDUT[uiLoopIterDMXDUTArraySeq] <> 0) THEN
		MEMCPY(srcAddr:=ADR(arruiDMXChDUT[uiLoopIterDMXDUTArraySeq]),destAddr:=ADR(arruiSeqTestIndicesTmp[uiLoopIterDMXDUTArraySeq]),n:=SIZEOF(arruiDMXChDUT[uiLoopIterDMXDUTArraySeq])); //UINT = 4 bytes?
//		uiLoopIterTestArrSeq		:= uiLoopIterTestArrSeq+1;
	END_IF
	uiLoopIterDMXDUTArraySeq	:= uiLoopIterDMXDUTArraySeq+1;
UNTIL 
(uiLoopIterDMXDUTArraySeq = gc.uiMaxNrOfDMXChannel)
END_REPEAT
//Stash the values from temp (inside FOR loop) to other arrays
arruiSeqTestIndices		:= arruiSeqTestIndicesTmp;

iSetConfig					:= 50;	

50:
//Use different iterators - set them to 0 prior to use
uiLoopIterDMXDUTArrayM		:= 0;
uiLoopIterTestArrM			:= 0;
//Zero out the array that is copied to in the next state of the SM
FOR uiForLoopZeroStorageArray	:= 0 TO gc.uiMaxNrOfDMXChannel BY 1 DO
	arruiMotorTestIndicesTmp[uiForLoopZeroStorageArray]	:= 0;
END_FOR
//Stash the values from temp (inside FOR loop) to other arrays
arruiMotorTestIndices	:= arruiMotorTestIndicesTmp;

iSetConfig					:= 60;	

60:
//Motors - Type code "M" - must be tested both in the PNP & NPN inputs
//This array easily provides the indexing for which channels the motors are on
REPEAT
	IF (arrsDUTChType[uiLoopIterDMXDUTArrayM] = 'M') AND (arruiDMXChDUT[uiLoopIterDMXDUTArrayM] <> 0)  THEN
		MEMCPY(srcAddr:=ADR(arruiDMXChDUT[uiLoopIterDMXDUTArrayM]),destAddr:=ADR(arruiMotorTestIndicesTmp[uiLoopIterDMXDUTArrayM]),n:=SIZEOF(arruiDMXChDUT[uiLoopIterDMXDUTArrayM])); //UINT = 4 bytes?
//		uiLoopIterTestArrM		:= uiLoopIterTestArrM+1;
	END_IF
	uiLoopIterDMXDUTArrayM	:= uiLoopIterDMXDUTArrayM+1;
UNTIL 
(uiLoopIterDMXDUTArrayM = gc.uiMaxNrOfDMXChannel)
END_REPEAT
//Stash the values from temp (inside FOR loop) to other arrays
arruiMotorTestIndices	:= arruiMotorTestIndicesTmp;

iSetConfig		:= 70;

70:
//Use different iterators - set them to 0 prior to use
uiLoopIterDUTArray24V		:= 0;
uiLoopIterTestArr24V		:= 0;
//Zero out the array that is copied to in the next state of the SM
FOR uiForLoopZeroStorageArray	:= 0 TO gc.uiMaxNrOfDMXChannel BY 1 DO
	arrui24VTestIndicesTmp[uiForLoopZeroStorageArray]	:= 0;
END_FOR
//Stash the values from temp (inside FOR loop) to other arrays
arrui24VTestIndices		:= arrui24VTestIndicesTmp;

iSetConfig				:= 80;

80:
//24V - Type code "24V" - is tested per static config
//This array easily provides the indexing for which channels the 24V are on
REPEAT
	IF (arrsDUTChType[uiLoopIterDUTArray24V] = '24V') AND (arruiDMXChDUT[uiLoopIterDUTArray24V] = 0) THEN
		MEMCPY(srcAddr:=ADR(arr_uiRecipeIndex[uiLoopIterDUTArray24V]),destAddr:=ADR(arrui24VTestIndicesTmp[uiLoopIterDUTArray24V]),n:=SIZEOF(arr_uiRecipeIndex[uiLoopIterDUTArray24V])); //UINT = 2 bytes?
//		uiLoopIterTestArr24V	:= uiLoopIterTestArr24V +1;
	END_IF
	uiLoopIterDUTArray24V	:= uiLoopIterDUTArray24V+1;
UNTIL 
(uiLoopIterDUTArray24V = gc.uiDUTConfigCountSplit)
END_REPEAT
//Stash the values from temp (inside FOR loop) to other arrays
arrui24VTestIndices	:= arrui24VTestIndicesTmp;

iSetConfig		:= 90;

90://Clear Iterators for GND channel indexing
//Use different iterators - set them to 0 prior to use
uiLoopIterDUTArrayGND		:= 0;
uiLoopIterTestArrGND		:= 0;
//Zero out the array that is copied to in the next state of the SM
FOR uiForLoopZeroStorageArray	:= 0 TO gc.uiMaxNrOfDMXChannel BY 1 DO
	arruiGNDTestIndicesTmp[uiForLoopZeroStorageArray]	:= 0;
END_FOR
//Stash the values from temp (inside FOR loop) to other arrays
arruiGNDTestIndices		:= arruiGNDTestIndicesTmp;

iSetConfig				:= 100;

100:
//Ground - Type code "GND" - is tested per static config
//This array easily provides the indexing for which channels the 24V are on
REPEAT
	IF (arrsDUTChType[uiLoopIterDUTArrayGND] = 'GND') AND (arruiDMXChDUT[uiLoopIterDUTArrayGND] = 0) THEN
		MEMCPY(srcAddr:=ADR(arr_uiRecipeIndex[uiLoopIterDUTArrayGND]),destAddr:=ADR(arruiGNDTestIndicesTmp[uiLoopIterDUTArrayGND]),n:=SIZEOF(arr_uiRecipeIndex[uiLoopIterDUTArrayGND])); //UINT = 4 bytes?
//		uiLoopIterTestArrGND	:= uiLoopIterTestArrGND+1;
	END_IF
	uiLoopIterDUTArrayGND	:= uiLoopIterDUTArrayGND+1;
UNTIL 
(uiLoopIterDUTArrayGND = gc.uiDUTConfigCountSplit)
END_REPEAT
//Stash the values from temp (inside FOR loop) to other arrays
arruiGNDTestIndices	:= arruiGNDTestIndicesTmp;

iSetConfig				:= 110;

//Copy of state30
110://Iterate over the config listings to create indices for what must be tested static (power, ground), and what must be tested sequentially (channels)
uiLoopIterDMXDUTArraySeq		:= 0;
uiLoopIterTestArrSeq			:= 0;
//Zero out the array that is copied to in the next state of the SM
FOR uiForLoopZeroStorageArray	:= 0 TO gc.uiMaxNrOfDMXChannel BY 1 DO
	arruiSeqTestIndicesDMXTmp[uiForLoopZeroStorageArray]	:= 0;
	arruiSeqTestIndicesDMXSW[uiForLoopZeroStorageArray]		:= 0;
END_FOR
//Stash the values from temp (inside FOR loop) to other arrays
arruiSeqTestIndicesDMX			:= arruiSeqTestIndicesDMXTmp;
iSetConfig						:= 120;	

120://Effectively a copy of state40
//For any 'DMX'-type channels with an assigned channel # (from the recipe), then copy only those elements to another array
//These are elements that are tested sequentially - once - so this includes Dry Contacts but not Motors
REPEAT
	IF (arrsDUTChType[uiLoopIterDMXDUTArraySeq] = 'DMX') AND (arruiDMXChDUT[uiLoopIterDMXDUTArraySeq] <> 0) THEN
		MEMCPY(srcAddr:=ADR(arruiDMXChDUT[uiLoopIterDMXDUTArraySeq]),destAddr:=ADR(arruiSeqTestIndicesDMXTmp[uiLoopIterDMXDUTArraySeq]),n:=SIZEOF(arr_uiRecipeIndex[uiLoopIterDUTArrayGND])); //UINT = 4 bytes?
//		uiLoopIterTestArrSeq		:= uiLoopIterTestArrSeq+1;
	END_IF
	uiLoopIterDMXDUTArraySeq		:= uiLoopIterDMXDUTArraySeq+1;
UNTIL 
(uiLoopIterDMXDUTArraySeq = gc.uiMaxNrOfDMXChannel)
END_REPEAT
//Stash the values from temp (inside FOR loop) to other arrays
arruiSeqTestIndicesDMX				:= arruiSeqTestIndicesDMXTmp;

//Set the recipe addresses one lower for 'SW'-Software-because software indexes from 0, not 1
FOR uiCounter8	:= 0 TO gc.uiMaxNrDMXTestCh BY 1 DO
	IF arruiSeqTestIndicesDMX[uiCounter8] <> 0 THEN
		arruiSeqTestIndicesDMXSW[uiCounter8]	:= arruiSeqTestIndicesDMX[uiCounter8] - 1;	
	END_IF
END_FOR

iSetConfig							:= 130;	

//Copy of state30
130://Iterate over the config listings to create indices for what must be tested static (power, ground), and what must be tested sequentially (channels)
uiLoopIterDMXDUTArraySeq		:= 0;
uiLoopIterTestArrSeq			:= 0;
//Zero out the array that is copied to in the next state of the SM
FOR uiForLoopZeroStorageArray	:= 0 TO gc.uiMaxNrOfDMXChannel BY 1 DO
	arruiSeqTestIndicesDCTmp[uiForLoopZeroStorageArray]	:= 0;
END_FOR
//Stash the values from temp (inside FOR loop) to other arrays
arruiSeqTestIndicesDC			:= arruiSeqTestIndicesDCTmp;
iSetConfig						:= 140;	

140:
//For any 'DMX'-type channels with an assigned channel # (from the recipe), then copy only those elements to another array
//These are elements that are tested sequentially - once - so this includes Dry Contacts but not Motors
REPEAT
	IF (arrsDUTChType[uiLoopIterDMXDUTArraySeq] = '24V') AND (arruiDMXChDUT[uiLoopIterDMXDUTArraySeq] <> 0) THEN
		MEMCPY(srcAddr:=ADR(arruiDMXChDUT[uiLoopIterDMXDUTArraySeq]),destAddr:=ADR(arruiSeqTestIndicesDCTmp[uiLoopIterDMXDUTArraySeq]),n:=SIZEOF(arruiDMXChDUT[uiLoopIterDMXDUTArraySeq])); //UINT = 4 bytes?
//		uiLoopIterTestArrSeq		:= uiLoopIterTestArrSeq+1;
	END_IF
	uiLoopIterDMXDUTArraySeq		:= uiLoopIterDMXDUTArraySeq+1;
UNTIL 
(uiLoopIterDMXDUTArraySeq = gc.uiMaxNrOfDMXChannel)
END_REPEAT
//Stash the values from temp (inside FOR loop) to other arrays
arruiSeqTestIndicesDC				:= arruiSeqTestIndicesDCTmp;

iSetConfig							:= 0;	

END_CASE


//Set the config of the 'routing' channels
IF r_tSetConfig.Q THEN
	g_ast.DMXHWOut	:= g_ast.DMXPhysOut;
//	xConfigSet		:= TRUE;
END_IF


// For manual setting of channels from the Visualization - NOTE! This stamps over any other values set for the lower 256 channels (DUT)
CASE iSetDUTSM OF
	
0:
IF r_tSetDUTVal.Q THEN
	iSetDUTSM		:= 10;
END_IF

10:
FOR uiForLoopDUTIter := 0 TO gc.uiDUTConfigCountSplit BY 1 DO
	g_ast.DMXHWOut[uiForLoopDUTIter] 	:= usiDUTVal;
END_FOR
//g_ast.DMXHWOut					:= g_ast.DMXPhysOut;

IF NOT r_tSetDUTVal.Q THEN
	iSetDUTSM	:= 0;
END_IF

END_CASE


CASE iSetExpctdBufferSM OF
	
0://If there is a trigger to set the test config, create a new 'Expctd' buffer
IF r_tSetExpectedBuff.Q THEN
	r_tExpectedBufferSet.CLK	:= FALSE;
	//Clear the existing buffers
	FOR uiForLoopClearExpctd := 0 TO gc.uiMaxNrOfDMXChannel BY 1 DO
		arrxExpctdPNP[uiForLoopClearExpctd]	:= 0;
		arrxExpctdNPN[uiForLoopClearExpctd]	:= 0;
	END_FOR
	iSetExpctdBufferSM			:= 10;
END_IF

10: // Set Expected Buffers per Recipe Files
FOR uiLoopExpctdIndex := 0 TO gc.uiMaxNrOfDMXChannel BY 1 DO
	IF (arr_usiRecipeSetting[uiLoopExpctdIndex] <= 127) THEN
		arrxExpctdPNP[arr_uiRecipeIndex[uiLoopExpctdIndex]]		:= TRUE; 
		arrxExpctdNPN[arr_uiRecipeIndex[uiLoopExpctdIndex]]		:= FALSE;
	ELSIF (arr_usiRecipeSetting[uiLoopExpctdIndex] > 127) THEN
		arrxExpctdPNP[arr_uiRecipeIndex[uiLoopExpctdIndex]]		:= FALSE;
		arrxExpctdNPN[arr_uiRecipeIndex[uiLoopExpctdIndex]]		:= TRUE; 
	END_IF
	//Zero out Expected, type-specific index buffers
	arrxExpctdTmpPNP24V[uiLoopExpctdIndex] 					:= 0;
	arrxExpctdTmpNPN24V[uiLoopExpctdIndex] 					:= 0;
	arrxExpctdTmpPNPGND[uiLoopExpctdIndex] 					:= 0;
	arrxExpctdTmpNPNGND[uiLoopExpctdIndex] 					:= 0;
END_FOR

r_tExpectedBufferSet.CLK	:= TRUE;
iSetExpctdBufferSM			:= 0;

END_CASE

CASE iReindexExpctedBufferSM OF
	
0:
IF r_tExpectedBufferSet.Q THEN
	iReindexExpctedBufferSM	:= 10;
END_IF

10://Copy the contents of Expected Buffer to a different Buffer, starting at array address 0 - only the channels that have a hardware input index
MEMCPY(srcAddr:=ADR(arrxExpctdPNP[gc.uiChannelSplitCount]),destAddr:=ADR(arrxExpctdTmpPNP[cuiMinDUTIndex]),n:=gc.uiChannelsUT);
MEMCPY(srcAddr:=ADR(arrxExpctdNPN[gc.uiChannelSplitCount]),destAddr:=ADR(arrxExpctdTmpNPN[cuiMinDUTIndex]),n:=gc.uiChannelsUT);

iReindexExpctedBufferSM	:= 20;

20:
//And create the comparison Expected Buffer for Static Test - 24V & GND indices
FOR uiCounter5 := 0 TO gc.uiMaxNrDMXTestCh BY 1 DO
	IF arrui24VTestIndices[uiCounter5] <> 0 THEN	
		MEMCPY(srcAddr:=ADR(arrxExpctdTmpPNP[arrui24VTestIndices[uiCounter5]]),destAddr:=ADR(arrxExpctdTmpPNP24V[arrui24VTestIndices[uiCounter5]]),n:=SIZEOF(arrxExpctdTmpPNP[arrui24VTestIndices[uiCounter5]])); //bytes
		MEMCPY(srcAddr:=ADR(arrxExpctdTmpNPN[arrui24VTestIndices[uiCounter5]]),destAddr:=ADR(arrxExpctdTmpNPN24V[arrui24VTestIndices[uiCounter5]]),n:=SIZEOF(arrxExpctdTmpNPN[arrui24VTestIndices[uiCounter5]])); //bytes
	END_IF
	
	IF arruiGNDTestIndices[uiCounter5] <> 0 THEN	
		MEMCPY(srcAddr:=ADR(arrxExpctdTmpPNP[arruiGNDTestIndices[uiCounter5]]),destAddr:=ADR(arrxExpctdTmpPNPGND[arruiGNDTestIndices[uiCounter5]]),n:=SIZEOF(arrxExpctdTmpPNP[arruiGNDTestIndices[uiCounter5]])); //bytes
		MEMCPY(srcAddr:=ADR(arrxExpctdTmpNPN[arruiGNDTestIndices[uiCounter5]]),destAddr:=ADR(arrxExpctdTmpNPNGND[arruiGNDTestIndices[uiCounter5]]),n:=SIZEOF(arrxExpctdTmpNPN[arruiGNDTestIndices[uiCounter5]])); //bytes
	END_IF	
END_FOR

iReindexExpctedBufferSM	:= 0;

END_CASE


CASE iCompareStaticSM OF
	
0: // If test is triggered by user
IF rt_RunStaticTest.Q THEN
	xStatTestInProgress						:= TRUE;
	uiLoopRcvIndex							:= cuiMinDUTIndex; 
	iCompareStaticSM						:= 10;
END_IF

10: // Zero out all comparison buffers before each comparison
//IF (uiLoopRcvIndex=0) THEN
	IF xStatTestInProgress THEN
		//by default, Counter = 0 at the first initialization; it is reset at the end of this State Machine
		//Clear Storage Buffers pre-test to ensure no old data interferes with current test
		FOR uiCounter4 := 0 TO gc.uiDUTConfigCountSplit BY 1 DO
			arrxRcvdBufferPNP24V[uiCounter4]	:= 0;		
			arrxRcvdBufferNPN24V[uiCounter4]	:= 0;		
			arrxRcvdBufferPNPGND[uiCounter4]	:= 0;		
			arrxRcvdBufferNPNGND[uiCounter4]	:= 0;
			gFB.arrFB_DMX[uiCounter4].I.xCmdOff	:= TRUE;		
//			g_ast.DMX[uiCounter4].IQ.xCmdOff	:= TRUE;	
		END_FOR
	iCompareStaticSM				:= 20;
	END_IF
(*
ELSIF (uiLoopRcvIndex>0) THEN
	IF xStatTestInProgress AND tonTestIterGap.Q THEN
		tonTestIterGap.IN	:= FALSE;
		//by default, Counter = 0 at the first initialization; it is reset at the end of this State Machine
		//Clear Storage Buffers pre-test to ensure no old data interferes with current test
		FOR uiCounter4 := 0 TO gc.uiDUTConfigCountSplit BY 1 DO
			arrxRcvdBufferPNP24V[uiCounter4]	:= 0;		
			arrxRcvdBufferNPN24V[uiCounter4]	:= 0;		
			arrxRcvdBufferPNPGND[uiCounter4]	:= 0;		
			arrxRcvdBufferNPNGND[uiCounter4]	:= 0;		
		END_FOR
	iCompareStaticSM				:= 30; // don't write the hardware value (skip 20)
	END_IF
END_IF
*)
	
20:	
//write 'hardware-clear' state 
g_ast.DMXHWOut					:= g_ast.DMXPhysOut;
iCompareStaticSM				:= 30;

30: //Set the Expected Mask & write data to controller
(*
IF uiLoopRcvIndex <> 0 THEN
//	g_ast.DMX[uiLoopRcvIndex].IQ.xCmdOn			:= TRUE;
	FOR uiCounter3 := cuiMinDUTIndex TO gc.uiMaxNrDMXTestCh BY 1 DO
		IF uiCounter3 <> uiLoopRcvIndex THEN
			g_ast.DMX[uiCounter3].IQ.xCmdOff	:= TRUE;	
		END_IF
	END_FOR
	iCompareStaticSM		:= 40;
ELSE //uiLoopRcvIndex = 0
	*)
tonWriteCopyWait.IN		:= TRUE;
iCompareStaticSM		:= 50;
//END_IF

40:
//Write DMX channels
(*
g_ast.DMXHWOut			:= g_ast.DMXPhysOut;
tonWriteCopyWait.IN		:= TRUE;
iCompareStaticSM		:= 50;
*)

50:
IF tonWriteCopyWait.Q THEN
	tonWriteCopyWait.IN	:= FALSE;
	iCompareStaticSM	:= 60;
END_IF

60:
FOR uiCounter4 := 0 TO gc.uiMaxNrDMXTestCh BY 1 DO

//IF there is an index for a '24V' element, then copy that element's value to a new pair of arrays, for 'Received'

	IF arrui24VTestIndices[uiCounter4] <> 0 THEN

		arrudiStaticCopyResultPNP24V[arrui24VTestIndices[uiCounter4]]	:= MEMCPY(srcAddr:=ADR(g_ast.arrInputPNP[arrui24VTestIndices[uiCounter4]]),destAddr:=ADR(arrxRcvdBufferPNP24V[arrui24VTestIndices[uiCounter4]]),n:=SIZEOF(g_ast.arrInputPNP[arrui24VTestIndices[uiCounter4]])); //bytes
		arrudiStaticCopyResultNPN24V[arrui24VTestIndices[uiCounter4]]	:= MEMCPY(srcAddr:=ADR(g_ast.arrInputNPN[arrui24VTestIndices[uiCounter4]]),destAddr:=ADR(arrxRcvdBufferNPN24V[arrui24VTestIndices[uiCounter4]]),n:=SIZEOF(g_ast.arrInputNPN[arrui24VTestIndices[uiCounter4]])); //bytes)

	END_IF

//IF there is an index for a 'GND' element, then copy that element's value to a new pair of arrays, for 'Received'

	IF arruiGNDTestIndices[uiCounter4] <> 0 THEN

		arrudiStaticCopyResultPNPGND[arruiGNDTestIndices[uiCounter4]]	:= MEMCPY(srcAddr:=ADR(g_ast.arrInputPNP[arruiGNDTestIndices[uiCounter4]]),destAddr:=ADR(arrxRcvdBufferPNPGND[arruiGNDTestIndices[uiCounter4]]),n:=SIZEOF(g_ast.arrInputPNP[arruiGNDTestIndices[uiCounter4]])); //bytes
		arrudiStaticCopyResultNPNGND[arruiGNDTestIndices[uiCounter4]]	:= MEMCPY(srcAddr:=ADR(g_ast.arrInputNPN[arruiGNDTestIndices[uiCounter4]]),destAddr:=ADR(arrxRcvdBufferNPNGND[arruiGNDTestIndices[uiCounter4]]),n:=SIZEOF(g_ast.arrInputNPN[arruiGNDTestIndices[uiCounter4]])); //bytes)
	
	END_IF
	
END_FOR

iCompareStaticSM			:= 70;

70:
tonReadWait.IN				:= TRUE;
iCompareStaticSM			:= 80;

80: // if wait completed, set the bit for conversion high
//Conversion Function call
IF tonReadWait.Q THEN
	tonReadWait.IN					:= FALSE;
	iCompareStaticSM				:= 90;
END_IF

90:
//Run Comparos
//Individual Channels comparison
FOR uiCounter6	:= 0 TO gc.uiMaxNrDMXTestCh BY 1 DO 
	arr_diTestStaticPNP24V[uiCounter6]		:= MEMCMP(pBuf1:=ADR(arrxExpctdTmpPNP24V[uiCounter6]),pBuf2:=ADR(arrxRcvdBufferPNP24V[uiCounter6]),n:=SIZEOF(arrxExpctdTmpPNP24V[uiCounter6]));
	arr_diTestStaticNPN24V[uiCounter6]		:= MEMCMP(pBuf1:=ADR(arrxExpctdTmpNPN24V[uiCounter6]),pBuf2:=ADR(arrxRcvdBufferNPN24V[uiCounter6]),n:=SIZEOF(arrxExpctdTmpNPN24V[uiCounter6]));
	arr_diTestStaticPNPGND[uiCounter6]		:= MEMCMP(pBuf1:=ADR(arrxExpctdTmpPNPGND[uiCounter6]),pBuf2:=ADR(arrxRcvdBufferPNPGND[uiCounter6]),n:=SIZEOF(arrxExpctdTmpPNPGND[uiCounter6]));
	arr_diTestStaticNPNGND[uiCounter6]		:= MEMCMP(pBuf1:=ADR(arrxExpctdTmpNPNGND[uiCounter6]),pBuf2:=ADR(arrxRcvdBufferNPNGND[uiCounter6]),n:=SIZEOF(arrxExpctdTmpNPNGND[uiCounter6]));
END_FOR

//Complete Buffer
diTestStaticPNP24V		:= MEMCMP(pBuf1:=ADR(arrxExpctdTmpPNP24V[cuiMinDUTIndex]),pBuf2:=ADR(arrxRcvdBufferPNP24V[cuiMinDUTIndex]),n:=gc.uiChannelsUT);
diTestStaticNPN24V		:= MEMCMP(pBuf1:=ADR(arrxExpctdTmpNPN24V[cuiMinDUTIndex]),pBuf2:=ADR(arrxRcvdBufferNPN24V[cuiMinDUTIndex]),n:=gc.uiChannelsUT);
diTestStaticPNPGND		:= MEMCMP(pBuf1:=ADR(arrxExpctdTmpPNPGND[cuiMinDUTIndex]),pBuf2:=ADR(arrxRcvdBufferPNPGND[cuiMinDUTIndex]),n:=gc.uiChannelsUT);
diTestStaticNPNGND		:= MEMCMP(pBuf1:=ADR(arrxExpctdTmpNPNGND[cuiMinDUTIndex]),pBuf2:=ADR(arrxRcvdBufferNPNGND[cuiMinDUTIndex]),n:=gc.uiChannelsUT);

iCompareStaticSM				:= 105;

(*
100: // If counter is equal to the max # of test channels, reset it; turn off the DMX channels that were turned on in the course of the test
IF (uiLoopRcvIndex = gc.uiMaxNrDMXTestCh) THEN
	rt_RunStaticTest.CLK			:= TRUE;
	iCompareStaticSM				:= 110;
ELSE
	uiLoopRcvIndex				:= uiLoopRcvIndex +1;
	//Next iteration
	tonTestIterGap.IN			:= TRUE;
	iCompareStaticSM			:= 10;
 (*iCounter <> gc.usiMaxNrOfChannels*)
END_IF
*)

105:
//Retrieving the discrepant indices for display on HMI
FOR uiVisuIndex := 0 TO gc.uiMaxNrDMXTestCh BY 1 DO
	IF (arr_diTestStaticPNP24V[uiVisuIndex] <> 0) THEN
		arrVisu_diTestResult[uiVisuIndex]	:= uiVisuIndex;	
	ELSIF (arr_diTestStaticNPNGND[uiVisuIndex] <> 0) THEN
		arrVisu_diTestResult[uiVisuIndex]	:= uiVisuIndex;	
	END_IF
END_FOR

iCompareStaticSM				:= 110;
	
110:
xStatTestInProgress				:= FALSE;
iCompareStaticSM				:= 120;

120:
IF rt_ResetTest.Q AND NOT rt_RunStaticTest.Q THEN
	FOR uiCounter2 := 0 TO gc.uiMaxNrDMXTestCh BY 1 DO 
		arr_diTestStaticPNP24V[uiCounter2]		:= 0;
		arr_diTestStaticNPN24V[uiCounter2]		:= 0;
		arr_diTestStaticPNPGND[uiCounter2]		:= 0;
		arr_diTestStaticNPNGND[uiCounter2]		:= 0;
	END_FOR
	diCompTestResult							:= 0;
	iCompareStaticSM							:= 0; (* reset to beginning *)
END_IF

END_CASE


//Linked to the Visualization Table
//FOR uiVisuIndex := 0 TO gc.uiMaxNrDMXTestCh BY 1 DO
	//	arrVisu_diTestResult[0,uiVisuIndex]	:= g_ast.DMXHWOut[uiVisuIndex]; //Sent
	//	arrVisu_diTestResult[1,uiVisuIndex]	:= arrbySclPNP[uiVisuIndex]; //Received
	//	arrVisu_diTestResult[2,uiVisuIndex]	:= arr_diTestResultPNP[uiVisuIndex]; //Result of Comparison
	//	arrVisu_diTestResult[3,uiVisuIndex]	:= arr_diTestResultNPN[uiVisuIndex]; //Result of Comparison
//END_FOR



//IF diCompTestResultTemp = -1 OR diCompTestResultTemp = 1 THEN
//	diCompTestResult	:= diCompTestResultTemp;
//END_IF

ACTION InvertRecipeSettings:
R_TInvertRecipe();

CASE iInvertRecipeSM OF
	
0:
IF R_TInvertRecipe.Q THEN
	iInvertRecipeSM		:= 10;
END_IF

10:
FOR uiRecipeInvertIter := uiStartingIndex TO uiEndingIndex BY 1 DO 
	IF arr_usiRecipeSetting[uiRecipeInvertIter] = 0 THEN
		arr_usiRecipeSetting[uiRecipeInvertIter]	:= 255;
	ELSIF arr_usiRecipeSetting[uiRecipeInvertIter] <> 0 THEN
		arr_usiRecipeSetting[uiRecipeInvertIter]	:= 0;
	END_IF
END_FOR

iInvertRecipeSM		:= 20;

20:
IF NOT R_TInvertRecipe.Q THEN
	iInvertRecipeSM		:= 0;
END_IF

END_CASE
END_ACTION

ACTION SeqTestMotor:

END_ACTION

ACTION SeqTestOnce:
//Run Once - DMX Channels only for now

rt_RunSeqTestOnce();
rt_ResetTestSeq();

CASE iCompareSeq[ENUM_SeqSM.Once] OF
	
0: // If test is triggered by user
//Trigger should be something like 
IF rt_RunSeqTestOnce.Q THEN
	xDMXSeqTestInProgressOnce				:= TRUE;
	uiLoopRcvIndex							:= cuiMinDUTIndex; 
	iCompareSeq[ENUM_SeqSM.Once]			:= 10;
END_IF

10: // Zero out all comparison buffers before each comparison
IF (uiLoopRcvIndex=0) THEN
	IF xDMXSeqTestInProgressOnce THEN
//by default, Counter = 0 at the first initialization; it is reset at the end of this State Machine
//Clear Storage Buffers pre-test to ensure no old data interferes with current test
		FOR uiCounter4 := 0 TO gc.uiMaxNrDMXTestCh BY 1 DO
			arrxExpctdTmpPNPSeqDMX[uiCounter4]		:= 0;		//should be all 0s ; PNP<>DMX
			arrxExpctdTmpNPNSeqDMX[uiCounter4]		:= 0;
//			arrxExpctdTmpPNPSeqDC[uiCounter4]		:= 0;		
//			arrxExpctdTmpNPNSeqDC[uiCounter4]		:= 0;
			arrxRcvdBufferPNPSeq[uiCounter4]		:= 0;		//should be all 0s too ; PNP<>DMX	
			arrxRcvdBufferNPNSeq[uiCounter4]		:= 0;
			gFB.arrFB_DMX[uiCounter4].I.xCmdOff	:= TRUE;				
		END_FOR
	iCompareSeq[ENUM_SeqSM.Once]					:= 20;
	END_IF
ELSIF (uiLoopRcvIndex>0) THEN // to avoid 
	IF xDMXSeqTestInProgressOnce AND tonTestIterGap.Q THEN
		tonTestIterGap.IN	:= FALSE;
		//by default, Counter = 0 at the first initialization; it is reset at the end of this State Machine
		//Clear Storage Buffers pre-test to ensure no old data interferes with current test
		FOR uiCounter4 := 0 TO gc.uiMaxNrDMXTestCh BY 1 DO
			arrxExpctdTmpPNPSeqDMX[uiCounter4]		:= 0;		//should be all 0s - PNP<>DMX
			arrxExpctdTmpNPNSeqDMX[uiCounter4]		:= 0;
			arrxRcvdBufferPNPSeq[uiCounter4]		:= 0;		
			arrxRcvdBufferNPNSeq[uiCounter4]		:= 0;
		END_FOR
		
	iCompareSeq[ENUM_SeqSM.Once]					:= 20; // don't write the hardware value (skip 20)
	END_IF	
END_IF
	
20:	
//write 'hardware-clear' state 
g_ast.DMXHWOut									:= g_ast.DMXPhysOut;

iCompareSeq[ENUM_SeqSM.Once]					:= 25;

25:
//Copy static test indices from Expected_Static - as these should still be used for comparisons
//	IF (arrui24VTestIndices[uiCounter4] <> 0) THEN	
//		MEMCPY(srcAddr:=ADR(arrxExpctdTmpPNP24V[cuiMinDUTIndex]),destAddr:=ADR(arrxExpctdTmpPNPSeqDMX[cuiMinDUTIndex]),n:=gc.uiChannelsUT);
FOR uiCounter4 := 0 TO gc.uiMaxNrDMXTestCh BY 1 DO
	arrxExpctdTmpPNPSeqDMX[uiCounter4]		:= arrxExpctdTmpPNP24V[uiCounter4];
	arrxExpctdTmpNPNSeqDMX[uiCounter4]		:= arrxExpctdTmpNPNGND[uiCounter4];
END_FOR

iCompareSeq[ENUM_SeqSM.Once]					:= 30;

30: //Set the Expected Mask & write data to controller
//Write the first index from the specified array of indices
//MEMCPY(srcAddr:=ADR(arrxExpctdTmpNPN[arruiSeqTestIndicesDMX[uiLoopRcvIndex]]),destAddr:=ADR(arrxExpctdTmpNPNSeqDMX[arruiSeqTestIndicesDMX[uiLoopRcvIndex]]),n:=SIZEOF(arrxExpctdTmpNPN[arruiSeqTestIndicesDMX[uiLoopRcvIndex]]));	

//This line copies only the value of the current iterator's index in the DMX Channel Array
arrxExpctdTmpNPNSeqDMX[uiLoopRcvIndex]	:= arrxExpctdTmpNPN[uiLoopRcvIndex];

iCompareSeq[ENUM_SeqSM.Once]			:= 35;

35:
IF (arruiSeqTestIndicesDMXSW[uiLoopRcvIndex] <> 0) THEN
//Also copy this specific channel index value to the comparison array
	
//Don't copy PNP indices for DMX; this doesn't generally make sense
//	MEMCPY(srcAddr:=ADR(arrxExpctdTmpPNP[arruiSeqTestIndicesDMX[uiLoopRcvIndex]]),destAddr:=ADR(arrxExpctdTmpPNPSeqDMX[arruiSeqTestIndicesDMX[uiLoopRcvIndex]]),n:=1);
	
	//CmdOn - command on - that respective channel
	gFB.arrFB_DMX[arruiSeqTestIndicesDMXSW[uiLoopRcvIndex]].I.xCmdOn			:= TRUE;
	//and turn off all others
	FOR uiCounter3 := cuiMinDUTIndex TO gc.uiMaxNrDMXTestCh BY 1 DO
		IF uiCounter3 <> arruiSeqTestIndicesDMXSW[uiLoopRcvIndex] THEN
			gFB.arrFB_DMX[uiCounter3].I.xCmdOff	:= TRUE;	
		END_IF
	END_FOR
END_IF

iCompareSeq[ENUM_SeqSM.Once]		:= 40;

40:
//Write to hardware
g_ast.DMXHWOut							:= g_ast.DMXPhysOut;
//tonWriteCopyWait.IN						:= TRUE;
iCompareSeq[ENUM_SeqSM.Once]			:=	60;

(*
50:

//Timer marks end of sampling period; reset timer
IF tonWriteCopyWait.Q THEN
	tonWriteCopyWait.IN					:=	FALSE;
	iCompareSeq[ENUM_SeqSM.Once]		:=	60;
END_IF
*)

60:
//Log all the 'gates' - returned from FB_Debounce
FOR uiCounter3	:= 0 TO gc.uiMaxNrDMXTestCh BY 1 DO
	arrxRcvdBufferNPNSeq[uiCounter3]		:= g_ast.arrFBIntNPN[uiCounter3].Q.xGate;
END_FOR
	
iCompareSeq[ENUM_SeqSM.Once]		:=	70;

//IF tonReadWait.Q THEN
//	tonReadWait.IN					:= FALSE;
//Copy hardware state
//	arrxRcvdBufferNPNSeq			:= arrxTestChInputNPN; // linked to hardware
//	arrxRcvdBufferPNPSeq			:= arrxTestChInputPNP; // linked to hardware
//iCompareSeq[ENUM_SeqSM.Once]		:= 90;
//END_IF

70:
//Run Comparos
//Individual
arr_diTestNPNSeqOnceLine[uiLoopRcvIndex]			:= MEMCMP(pBuf1:=ADR(arrxExpctdTmpNPNSeqDMX[uiLoopRcvIndex]),pBuf2:=ADR(arrxRcvdBufferNPNSeq[uiLoopRcvIndex]),n:=SIZEOF(arrxExpctdTmpNPNSeqDMX[uiLoopRcvIndex])); 
//Complete Buffer
arrdiTestNPNSeqOnceComplete[uiLoopRcvIndex]			:= MEMCMP(pBuf1:=ADR(arrxExpctdTmpNPNSeqDMX[cuiMinDUTIndex]),pBuf2:=ADR(arrxRcvdBufferNPNSeq[cuiMinDUTIndex]),n:=gc.uiChannelsUT); 

//log the error index - later

iCompareSeq[ENUM_SeqSM.Once]				:= 80;

80: //Turn off all DMX channels after comparison
FOR uiCounter3 := cuiMinDUTIndex TO gc.uiMaxNrDMXTestCh BY 1 DO
	gFB.arrFB_DMX[uiCounter3].I.xCmdOff		:= TRUE;
END_FOR

90://Write to DMX hardware, advance state
g_ast.DMXHWOut								:= g_ast.DMXPhysOut;

iCompareSeq[ENUM_SeqSM.Once]				:= 100;

100: //Confirm 'return' to static 
FOR uiCounter3	:= 0 TO gc.uiMaxNrDMXTestCh BY 1 DO
	arrxRcvdBufferNPNSeq[uiCounter3]		:= g_ast.arrFBIntNPN[uiCounter3].Q.xGate;
	IF arrxRcvdBufferNPNSeq[uiCounter3] = arrxExpctdTmpNPNGND[uiCounter3] THEN
		iCompareSeq[ENUM_SeqSM.Once]				:= 110;
	END_IF
END_FOR

110://Write to DMX hardware, advance state
g_ast.DMXHWOut								:= g_ast.DMXPhysOut;

iCompareSeq[ENUM_SeqSM.Once]				:= 120;

120: // If counter is equal to the max # of test channels, reset it; else, proceed around again 
IF (uiLoopRcvIndex = gc.uiMaxNrDMXTestCh) THEN
	iCompareSeq[ENUM_SeqSM.Once]			:= 130;
ELSE
	uiLoopRcvIndex							:= uiLoopRcvIndex +1;
	//Next iteration
	tonTestIterGap.IN						:= TRUE;
	iCompareSeq[ENUM_SeqSM.Once]			:= 10;
 (*iCounter <> gc.usiMaxNrOfChannels*)
END_IF

130:
xDMXSeqTestInProgressOnce					:= FALSE;
iCompareSeq[ENUM_SeqSM.Once]				:= 140;

140:
IF rt_ResetTestSeq.Q AND NOT rt_RunSeqTestOnce.Q THEN
	FOR uiCounter2 := 0 TO gc.uiMaxNrDMXTestCh BY 1 DO 
		arr_diTestPNPSeqOnceLine[uiCounter2]		:= 0;
		arr_diTestNPNSeqOnceLine[uiCounter2]		:= 0;
//		arrdiTestPNPSeqOnceComplete[uiCounter2]		:= 0;
//		arrdiTestNPNSeqOnceComplete[uiCounter2]		:= 0;
		arrdiTestNPNSeqOnceCompleteProblemIndex[uiCounter2]	:= 0;
	END_FOR
	diCompTestResult							:= 0;
	iCompareSeq[ENUM_SeqSM.Once]				:= 0; (* reset to beginning *)
END_IF

END_CASE
END_ACTION

ACTION SeqTestOnceDC:

END_ACTION

END_PROGRAM

// ---- POUs/P_TextModeRead.TcPOU
(* Reading of CSV file in text mode. None of the field value is containing any non-printing control characters like line feed, carriage return, quotation marks, semicolon... *)
PROGRAM P_TextModeRead
VAR
	bRead			: BOOL := FALSE;(* Rising edge starts program execution *)
	sNetId			: T_AmsNetId := '';	(* TwinCAT system network address *)
	sFileName		: T_MaxString;(* CSV source file path and name *)
	sCSVLine		: T_MaxString := '';(* Single CSV text line (row, record), we are using string as record buffer (your are able to see read fields)  *)
	sCSVField		: T_MaxString := '';(* Single CSV field value (column, record field) *)
	bBusy			: BOOL;
	bError			: BOOL;
	nErrId			: UDINT;
	nRow	 		: UDINT 	:= 0;(* Row number (record) *)
	nColumn			: UDINT 	:= 0;(* Column number (record field) *)
	hFile			: UINT		:= 0;(* File handle of the source file *)
	step			: DWORD 	:= 0;
	fbFileOpen		: FB_FileOpen;(* Opens file *)
	fbFileClose		: FB_FileClose;(* Closes file *)
	fbFileGets		: FB_FileGets;(* Reads one record (line) *)
	fbReader		: FB_CSVMemBufferReader;(* Helper function block used to parse CSV data bytes (single record line) *)
	database		: ARRAY[0..MAX_CSV_ROWS, 0..MAX_CSV_COLUMNS ] OF STRING(MAX_CSV_FIELD_LENGTH);(* Target PLC database *)
	sFileNameQueued	: STRING(255);
	sFilePathHMI	: STRING(255);
	r_tFileChg		: R_TRIG;
END_VAR

CASE step OF
	0:	(* Wait for rising edge at bRead variable *)
		IF bRead THEN
			bRead 	:= FALSE;
			bBusy 	:= TRUE;
			bError	:= FALSE;
			nErrId	:= 0;
			hFile	:= 0;
			nRow	:= 0;
			nColumn	:= 0;
			MEMSET( ADR( database ), 0, SIZEOF( database ) );
			step 		:= 1;
		END_IF

	1:	(* Open source file *)
		fbFileOpen(  bExecute := FALSE  );
		fbFileOpen( sNetId := sNetId, sPathName := sFileName, nMode := FOPEN_MODEREAD OR FOPEN_MODETEXT,(* Open file in TEXT mode! *)
					ePath := PATH_GENERIC, bExecute := TRUE );
		step := 2;

	2:(* Wait until open not busy *)
		fbFileOpen( bExecute := FALSE, bError => bError, nErrID => nErrID, hFile => hFile );
		IF NOT fbFileOpen.bBusy THEN
			IF NOT fbFileOpen.bError THEN
				step := 3;
			ELSE(* Error: file not found? *)
				step := 100;
			END_IF
		END_IF

	3:	(* Read single line (record) *)
		fbFileGets( bExecute := FALSE );
		fbFileGets( sNetId := sNetId, hFile := hFile, bExecute := TRUE );
		step := 4;

	4:(* Wait until read not busy *)
		fbFileGets( bExecute := FALSE, bError => bError, nErrID => nErrID, sLine => sCSVLine );
		IF NOT fbFileGets.bBusy THEN
			IF NOT fbFileGets.bError THEN
				IF fbFileGets.bEOF THEN
					step := 10;(* End of file reached => Close source file *)
				ELSE

					(* FB_FileGets returns text line without the CR (carriage return) character.
					We have to restore the CR character (replace the $L character with $R$L characters) *)
					IF RIGHT( sCSVLine, 1 ) = '$L' THEN
						sCSVLine := REPLACE( sCSVLine, '$R$L', 2, LEN( sCSVLine ) );
					END_IF

					step := 5;
				END_IF
			ELSE(* Error *)
				step := 100;
			END_IF
		END_IF

	5:(* Parse single line (record) *)
		fbReader.eCmd := eEnumCmd_First;(* Read first field value *)
		REPEAT
			fbReader( pBuffer := ADR( sCSVLine ), cbBuffer := SIZEOF( sCSVLine ), getValue => sCSVField );
			IF fbReader.bOk THEN
				fbReader.eCmd := eEnumCmd_Next;(* Read next field value *)

				IF ( nRow <= MAX_CSV_ROWS ) THEN
					IF ( nColumn <= MAX_CSV_COLUMNS ) THEN
						database[nRow, nColumn] := CSVFIELD_TO_STRING( sCSVField, FALSE );(* TODO: Save or use the field value in your application *)
					END_IF
				END_IF

				nColumn := nColumn + 1;(* Increment number of read columns *)
				IF fbReader.bCRLF THEN(* CRLF == TRUE => End of reacord reached *)
					nRow 		:= nRow + 1;(* Increment number of read records *)
					nColumn 	:= 0;(* Reset number of columns *)
				END_IF

			ELSE(* Error: End of record reached or all fields read *)
				step := 3;(* Try to read next line *)
			END_IF
		UNTIL NOT fbReader.bOk
		END_REPEAT

	10:	(* Close source file *)
		fbFileClose( bExecute := FALSE );
		fbFileClose( sNetId := sNetId, hFile := hFile, bExecute := TRUE );
		step := 11;

	11:(* Wait until close not busy *)
		fbFileClose( bExecute := FALSE, bError => bError, nErrID => nErrID );
		IF ( NOT fbFileClose.bBusy ) THEN
			hFile := 0;
			step := 100;
		END_IF

	100: (* Error or ready step => cleanup *)
		IF ( hFile <> 0 ) THEN
			step := 10; (* Close the source file *)
		ELSE
			bBusy := FALSE;
			step := 0;	(* Ready *)
		END_IF

END_CASE

sFileNameQueued	:= sFilePathHMI	;
r_tFileChg();
bRead	:= r_tFileChg.CLK;

IF r_tFileChg.Q THEN
	sFileName	:= sFileNameQueued;
END_IF

END_PROGRAM

// ---- POUs/DMXShop.TcPOU
PROGRAM DMXShop
VAR
	afbDMXRGBW	: ARRAY[0..3] OF FBOscillator;
	iforloop	: INT;
END_VAR

//afbDMXRGBW[gc.RED].I.ENWaveform			:= ENUM_I_Waveform.EN_Triangle; //"50% duty cycle"
//afbDMXRGBW[gc.RED].I.fDutyCycle			:= 50; // %
//afbDMXRGBW[gc.RED].I.fLevel				:= 100; //%
//afbDMXRGBW[gc.RED].I.fOffset			:= 0; // %
//afbDMXRGBW[gc.RED].I.usiBitDepth		:= 8; // 0-8, or 0-16, depending
//afbDMXRGBW[gc.RED].I.fPhase				:= 0; // %
//afbDMXRGBW[gc.RED].I.fDelay				:= 0; // %
//afbDMXRGBW[gc.RED].I.usiDelayDiv		:= 0; // which step to have delay applied
//afbDMXRGBW[gc.RED].I.fFrequency			:= 50;

//afbDMXRGBW[gc.GREEN].I.ENWaveform		:= ENUM_I_Waveform.EN_Triangle; //"50% duty cycle"
//afbDMXRGBW[gc.GREEN].I.fDutyCycle		:= 50; // %
//afbDMXRGBW[gc.GREEN].I.fLevel			:= 100; //%
//afbDMXRGBW[gc.GREEN].I.fOffset			:= 0; // %
//afbDMXRGBW[gc.GREEN].I.usiBitDepth		:= 8; // 0-8, or 0-16, depending
//afbDMXRGBW[gc.GREEN].I.fPhase			:= 0; // %
//afbDMXRGBW[gc.GREEN].I.fDelay			:= 0; // %
//afbDMXRGBW[gc.GREEN].I.usiDelayDiv		:= 0; // which step to have delay applied
//afbDMXRGBW[gc.GREEN].I.fFrequency		:= 50; 

//afbDMXRGBW[gc.BLUE].I.ENWaveform		:= ENUM_I_Waveform.EN_Triangle; //"50% duty cycle"
//afbDMXRGBW[gc.BLUE].I.fDutyCycle		:= 50; // %
//afbDMXRGBW[gc.BLUE].I.fLevel			:= 100; //%
//afbDMXRGBW[gc.BLUE].I.fOffset			:= 0; // %
//afbDMXRGBW[gc.BLUE].I.usiBitDepth		:= 8; // 0-8, or 0-16, depending
//afbDMXRGBW[gc.BLUE].I.fPhase			:= 0; // %
//afbDMXRGBW[gc.BLUE].I.fDelay			:= 0; // %
//afbDMXRGBW[gc.BLUE].I.usiDelayDiv		:= 0; // which step to have delay applied
//afbDMXRGBW[gc.BLUE].I.fFrequency		:= 50;

//afbDMXRGBW[gc.WHITE].I.ENWaveform		:= ENUM_I_Waveform.EN_Triangle; //"50% duty cycle"
//afbDMXRGBW[gc.WHITE].I.fDutyCycle		:= 50; // %
//afbDMXRGBW[gc.WHITE].I.fLevel			:= 100; //%
//afbDMXRGBW[gc.WHITE].I.fOffset			:= 0; // %
//afbDMXRGBW[gc.WHITE].I.usiBitDepth		:= 8; // 0-8, or 0-16, depending
//afbDMXRGBW[gc.WHITE].I.fPhase			:= 0; // %
//afbDMXRGBW[gc.WHITE].I.fDelay			:= 0; // %
//afbDMXRGBW[gc.WHITE].I.usiDelayDiv		:= 0; // which step to have delay applied
//afbDMXRGBW[gc.WHITE].I.fFrequency		:= 50; 

afbDMXRGBW[gc.RED].tPeriodRise		:= T#80S;
afbDMXRGBW[gc.GREEN].tPeriodRise	:= T#130S;
afbDMXRGBW[gc.BLUE].tPeriodRise		:= T#210S;
afbDMXRGBW[gc.WHITE].tPeriodRise	:= T#10S;

afbDMXRGBW[gc.RED].tPeriodFall		:= T#13S;
afbDMXRGBW[gc.GREEN].tPeriodFall	:= T#13S;
afbDMXRGBW[gc.BLUE].tPeriodFall		:= T#11S;
afbDMXRGBW[gc.WHITE].tPeriodFall	:= T#340S;

FOR iforloop := 0 TO gc.WHITE BY 1 DO
	afbDMXRGBW[iforloop]();
END_FOR

END_PROGRAM

// ---- POUs/FBOscillator.TcPOU
FUNCTION_BLOCK FBOscillator
VAR_INPUT
	tPeriodRise	: TIME;
	tPeriodFall	: TIME;
END_VAR
VAR_OUTPUT
	byValue	 AT %Q*	: BYTE;
END_VAR
VAR
	tonRise	: TON;
	tonFall : TON;
	MAXVALUE	: UDINT := 255;
	iCycle  : INT;
END_VAR

tonRise(PT	:= tPeriodRise);
tonFall(PT	:= tPeriodFall);

CASE iCycle OF
	
0:
tonRise.IN	:= TRUE;
iCycle		:= 10;

10:
IF tonRise.Q THEN
	tonRise.IN	:= FALSE;
	tonFall.IN	:= TRUE;
	iCycle		:= 20;
END_IF

20:
IF tonFall.Q THEN
	tonFall.IN	:= FALSE;
	iCycle		:= 0;
END_IF

END_CASE

IF tonRise.IN THEN
	byValue	:= UDINT_TO_BYTE(MAXVALUE);
ELSE
	byValue	:= 3;
END_IF

END_FUNCTION_BLOCK

// ---- POUs/FB_DMX.TcPOU
FUNCTION_BLOCK FB_DMX
VAR_INPUT
	I	: typDMXInput;
END_VAR

//VAR_IN_OUT
//	I	: typDMXInOut;
//END_VAR

VAR_OUTPUT
	Q	AT %Q* : typDMXOutput;
END_VAR

VAR
//	uiOpStatus			: UINT;
	iWaveSelectSM		: INT;
	uiTimeCycleSM		: UINT;
	uiDelayShiftSM		: UINT;
	uiTimeShiftSM		: UINT;
	uiDeviceSM			: UINT;
	uiModeCtrlSM		: UINT;

	uiPulseCount		: UINT;
	fPhaseShift			: REAL;
	fDelayShift			: REAL;
	tTimeShift			: TIME;
	tPhaseShift			: TIME;
	tDelayShift			: TIME;

	fLevelShift			: REAL;
	fOffsetShift		: REAL;	
	tOnPulse			: TON;
	tOnShift			: TON;
	
	tonFnWindow			: TON;
	tonSqDutyCyc		: TON;
	fDutyCycle			: REAL;
	
	fFnGenerValTempSin	: LREAL;
	fFnGenerValAdj		: REAL; //Adjusted channel value: rounded, clamped, scaled per the input parameters for the channel
	
	rt_FnRisEdge		: R_TRIG;
	
	cfLoFnVal			: REAL	:= 0; // min function value from function generator
	cfHiFnVal			: REAL	:= 2; // max function value from function generator
	
	fFnWindowET			: REAL;
	tPeriod				: TIME;
	tonRunning			: TON;
	tonRunningSH		: TON;
	iClockSM			: INT;
	iFnSampleHoldSM		: INT;
	
	//not currently used:	
	tonFnSomethingElse	: TON;
	
	fPeriod				: REAL;
	tFnWindowET			: TIME;
END_VAR

//Compute Regular Trigger/Pulse train:
CASE uiTimeCycleSM OF
	
0: //Execute timer
tOnPulse.IN		:= TRUE;
uiTimeCycleSM	:= 10;

10:  //Wait for timer completion ; reset timer
IF tOnPulse.Q THEN
	tOnPulse.IN		:= FALSE;
	uiTimeCycleSM	:= 0;
END_IF

END_CASE

//calculate time shift
tPhaseShift	:= REAL_TO_TIME(fPhaseShift);

tDelayShift	:= REAL_TO_TIME(fDelayShift);

tTimeShift	:= tPhaseShift + tDelayShift;

//Phase Shift Function
fPhaseShift	:= (I.fPhase/100)(*percentage*)*fPeriod;

//Delay Shift also uses this SM (State Machine) in order to apply fDelayShift on the appropriate step
CASE uiDelayShiftSM OF
	
0:
IF tOnPulse.Q THEN
	uiPulseCount	:= uiPulseCount + 1;
	uiDelayShiftSM	:= 10;
END_IF

10: // State to apply the Delay Time Shift

//Reset the Pulse Counter if it is equivalent to the delay divisor ; and shift state to apply the delay on that "step"
IF uiPulseCount = I.usiDelayDiv THEN
	uiPulseCount	:= 0;
	//Delay Shift Function
	IF I.fFrequency <> 0 THEN
		fDelayShift	:= (I.fDelay/100)(*percentage*)*fPeriod;
	END_IF
ELSIF (I.usiDelayDiv = 0) THEN
	uiPulseCount	:= 0;
ELSE (* uiPulseCount <> I.usiDelayDiv THEN *)  
	fDelayShift		:= 0; (* Delay Shift always = 0 when it is on a step that is not equal to I.usiDelayDiv *)
	uiDelayShiftSM	:= 0; (* return to increment pulse counter *)
END_IF

END_CASE

//This SM sees rising edge from pulse; applies time shift (even if time shift = 0)
CASE uiTimeShiftSM OF 
	
0: // If there is a rising edge from the Pulse clock, implement tonShift, a delay
IF tOnPulse.IN THEN
	tOnShift.IN	:= TRUE;
	uiTimeShiftSM	:= 10;
END_IF

10:
IF tOnShift.Q THEN
	tOnShift.IN		:= FALSE;
	uiTimeShiftSM	:= 0;
END_IF

END_CASE


//level shift code:
//offset adjusts 'bottom' rail, level adjusts 'top' rail;
//bit depth specifies the 'fine-ness' of the value range for the output
//Sets the I - basically modifies the user input 'I'

IF I.ENValRange = ENUM_I_ValRange.EN_8Bit THEN //accept the user input params
	I.uiMaxChannelVal	:= 255;
ELSIF I.ENValRange = ENUM_I_ValRange.EN_16Bit THEN //accept the user input params
	I.uiMaxChannelVal	:= 65535;
END_IF

//perhaps have a 'preset' condition like this, for Boolean:
//Sets the I - basically modifies the user input 'I'
IF (I.ENWaveform = ENUM_I_Waveform.EN_GateCtrl) OR (I.ENWaveform = ENUM_I_Waveform.EN_GateConfig) OR (I.usiBitDepth = 1) THEN
	I.fLevel		:= Map(fArg:=100(*%*),fInMin:=0,fInMax:=100,fOutMin:=I.uiMinChannelVal,fOutMax:=I.uiMaxChannelVal);
	I.usiBitDepth	:= 1;
	I.fOffset		:= Map(fArg:=0(*%*),fInMin:=0,fInMax:=100,fOutMin:=I.uiMinChannelVal,fOutMax:=I.uiMaxChannelVal);
ELSE (* not Boolean/Gate operation *)
	I.fLevel		:= Map(I.fLevel,0,100,0,I.uiMaxChannelVal); // scale % to 255
	I.usiBitDepth	:= I.usiBitDepth; 
	I.fOffset		:= Map(I.fOffset,0,100,0,I.uiMaxChannelVal); // scale % to 255
END_IF

//Return a mapped value, clamped to a 'nearest value' governed by the bit depth
//Check I.fFnGenerValRtn range; if it's from the sin function, use input range [0,2]; else use [0,100]

Q.byStatValue		:= REAL_TO_BYTE(Q.fFnGeneratorVal);
I.byMinChanVal		:= UINT_TO_BYTE(I.uiMinChannelVal);
I.byMaxChanVal		:= UINT_TO_BYTE(I.uiMaxChannelVal);

tFnWindowET			:= tonRunning.ET;
fFnWindowET			:= TIME_TO_REAL(tFnWindowET);

CASE iWaveSelectSM OF

// Wave Select State Machine needs to output a "function" value.  This can be continuously generated.  In all cases, let's say for example's sake we are using something like "f(x) = sin(x)".  
// The values of the function output should be scaled from (0,2) of (-1,1).  The scaled value should be input to the function below that maps and re-scales this function output, 
// to fit the range of user parameters (level, offset, bit depth) specified.  Perhaps this for all function outputs - 

0: // Default to zero state for this SM, then go to the relevant function generator (enumerator) state
IF rt_FnRisEdge.Q THEN
	tonFnWindow.IN	:= TRUE;
	iWaveSelectSM	:= I.ENWaveform;
END_IF

ENUM_I_Waveform.EN_Square:
IF I.fFrequency = 0 THEN
	I.fFnGenerValRtn	:= I.fLevel; // Set it to the permissible max of the range
ELSE (* I.fFrequency <> 0 *)
	tonSqDutyCyc.IN		:= TRUE;
	I.fFnGenerValRtn	:= 255*BOOL_TO_LREAL(tonSqDutyCyc.IN);
	iWaveSelectSM		:= 15;
END_IF

15:
IF tonSqDutyCyc.Q THEN
	tonSqDutyCyc.IN		:= FALSE;
	iWaveSelectSM		:= ENUM_I_Waveform.EN_Square;
END_IF

//Basically the same as 'Square' but no 'duty cycle'
ENUM_I_Waveform.EN_GateConfig (* Note 8-bit Only *):

// Relay NC condition = PNP; Relay 'NO' condition = NPN
// Otherwise, DMX Function Block should function normally
IF (I.usiInputConfig <= (0.5*I.uiMaxChannelVal)) THEN
	I.fFnGenerValRtn		:= I.fOffset;
ELSIF (I.usiInputConfig > (0.5*I.uiMaxChannelVal)) THEN
	I.fFnGenerValRtn		:= I.fLevel;
END_IF

Q.fFnGeneratorVal		:= I.fFnGenerValRtn; // Set it to the permissible max of the range

ENUM_I_Waveform.EN_GateCtrl:
IF I.xCmdOn THEN
	I.xCmdOn			:= FALSE;
	I.fFnGenerValRtn	:= I.fLevel;
END_IF

IF I.xCmdOff THEN
	I.xCmdOff			:= FALSE;
	I.fFnGenerValRtn	:= I.fOffset;
END_IF

Q.fFnGeneratorVal		:= I.fFnGenerValRtn; // Set it to the permissible max of the range

ENUM_I_Waveform.EN_Sin:
IF I.ENWaveform = ENUM_I_Waveform.EN_Sin THEN
	Q.fFnGeneratorVal		:= MapClamp(I.fFnGenerValRtn,cfLoFnVal,cfHiFnVal,I.fOffset,I.fLevel,I.usiBitDepth);
ELSE
	Q.fFnGeneratorVal		:= MapClamp(I.fFnGenerValRtn,I.fOffset,I.fLevel,I.fOffset,I.fLevel,I.usiBitDepth);
END_IF

tFnWindowET			:= tonRunning.ET;
fFnWindowET			:= TIME_TO_REAL(tFnWindowET);

I.fFnGenerValTempSin	:= (2*gc.fPi*I.fFrequency*fFnWindowET);

//y(t)=sin(2*pi*f*t)
(*
CASE iFnSampleHoldSM OF
	
0:
tonRunningSH.IN		:= TRUE;
iFnSampleHoldSM		:= 10;

10:
IF tonRunningSH.Q THEN
	tonRunningSH.IN		:= FALSE;
	tFnWindowET			:= tonRunning.ET;
	fFnWindowET			:= TIME_TO_REAL(tFnWindowET);
	iFnSampleHoldSM	:= 0;
END_IF

END_CASE
*)

ENUM_I_Waveform.EN_Triangle:
Q.fFnGeneratorVal	:= 2; //set function value high initially, advance SM

iWaveSelectSM		:= ENUM_I_Waveform.EN_SubTriFall;

ENUM_I_Waveform.EN_SubTriFall:

//use 2 as the function value (that is the range of the function)
IF fPeriod <> 0 THEN
	Q.fFnGeneratorVal	:= Q.fFnGeneratorVal - ((2 / (fPeriod*0.5))*fFnWindowET);
END_IF

IF Q.fFnGeneratorVal = 0 THEN
	iWaveSelectSM		:= ENUM_I_Waveform.EN_SubTriRise;
END_IF

//use 2 as the function value (that is the range of the function)
ENUM_I_Waveform.EN_SubTriRise:
IF fPeriod <> 0 THEN
	Q.fFnGeneratorVal	:= Q.fFnGeneratorVal + ((2 / (fPeriod*0.5))*fFnWindowET);
END_IF

IF Q.fFnGeneratorVal = 2 THEN
	iWaveSelectSM		:= ENUM_I_Waveform.EN_Triangle;
END_IF
	
END_CASE
	
//ENUM_I_Waveform.EN_Ramp:
//function output range from (0,255) - level/offset/depth transformation (for scaling) happens separately

//ENUM_I_Waveform.EN_Rand:
//function output range from (0,255) - level/offset/depth transformation (for scaling) happens separately

//ENUM_I_Waveform.EN_Saw:
//function output range from (0,255) - level/offset/depth transformation (for scaling) happens separately

(*
CASE uiModeCtrlSM OF
	
//ENUM_I_OpMode.EN_Cycle:

ENUM_I_OpMode.EN_Cycle:


ENUM_I_OpMode.EN_LatchOn:

ENUM_I_OpMode.EN_OneShot:


END_CASE*)

//crufty - may be useful in future cleaning up of this FB, or not
(*
ELSIF Q.xGate (* or Function Output *) THEN
	Q.byStatValue		:= REAL_TO_BYTE(Q.fFnGeneratorVal);
ELSE (*<> Q.xGate*) (* "Offset" equivalent to the 'recipe'-adjusted 'zero' *)
	Q.byStatValue		:= REAL_TO_BYTE(I.fOffset);	
END_IF
*)


CASE iClockSM OF
	
0: // Start clock
tonRunning.IN	:= TRUE;
iClockSM	:= 10;

10:
IF tonRunning.Q THEN
	tonRunning.IN	:= FALSE;
	iClockSM		:= 0;
END_IF

END_CASE

IF I.fFrequency <> 0 THEN
	fPeriod		:= f_to_Period(I.fFrequency);
END_IF

tPeriod			:= REAL_TO_TIME(1000*fPeriod);

//Function Calls / Parameterization
rt_FnRisEdge(CLK	:= tOnShift.IN);
tOnPulse();
tOnPulse.PT		:= tPeriod;
tOnShift(PT	:= tTimeShift / 2);

//tonFnSomethingElse(PT	:= (REAL_TO_TIME(f_to_Period(I.fFrequency)) - tOnPulse.PT - tOnShift.PT (*- T#1MS*))); // Used for cycle mode; cycle should reset before the next 'pulse' occurs
tonFnWindow(PT	:= tPeriod); // Only dependent on period

IF I.fFrequency <> 0 THEN
	fDutyCycle	:= ((I.fDutyCycle/100) * TIME_TO_REAL(tonFnWindow.PT)); // % of the time window that the value is to be held high	
END_IF
tonSqDutyCyc();
tonSqDutyCyc.PT	:= REAL_TO_TIME(fDutyCycle);
tonRunning(PT	:= T#24H);
tonRunningSH(PT	:= T#1MS); // Preset time for how quickly to sample the ET value from 'tonRunning' - how quickly does SIN "Sample & Hold" function refresh?

END_FUNCTION_BLOCK

// ---- POUs/FB_InputDebounce.TcPOU
FUNCTION_BLOCK FB_InputDebounce
VAR_INPUT
	I	: typFBDInput;
END_VAR

VAR_IN_OUT
	IQ	: typFBDInOut;
END_VAR

VAR_OUTPUT
	Q	: typFBDOutput;
END_VAR

VAR
	tonOnDelay		: TON;
	tofOffDelay		: TOF;
	uiDebounceSM	: UINT;
END_VAR

tonOnDelay(PT	:= I.tOnDelay);
tofOffDelay(PT	:= I.tOffDelay);

CASE uiDebounceSM OF
	
0: // If there is a trig, then set a timer for the On Delay
IF IQ.xTrig THEN
	tonOnDelay.IN	:= TRUE;
	tofOffDelay.IN	:= TRUE;
	uiDebounceSM	:= 10;
END_IF

10: // If timer is completed, set the timer false, set the Gate (output) high, falling edge to TOF input
IF tonOnDelay.Q THEN
	tonOnDelay.IN	:= FALSE;
	Q.xGate			:= TRUE;
	tofOffDelay.IN	:= FALSE;
	uiDebounceSM	:= 20;	
END_IF

20: // Falling edge on TOF drops Gate
IF NOT tofOffDelay.Q AND NOT IQ.xTrig THEN
	Q.xGate			:= FALSE;
	uiDebounceSM	:= 30;
ELSIF NOT tofOffDelay.Q AND IQ.xTrig THEN
//Jump state; no other actions (do not set gate false)
	uiDebounceSM	:= 40;
END_IF

30: //Ensure the trig has gone low
IF NOT IQ.xTrig THEN
	uiDebounceSM	:= 0;
END_IF

40: // State for "if trig held past OffDelay time"; if trig has gone low, set gate low
IF NOT IQ.xTrig THEN
	Q.xGate			:= FALSE;
	uiDebounceSM	:= 0;
END_IF
	
END_CASE

END_FUNCTION_BLOCK

// ---- POUs/MAIN.TcPOU
PROGRAM MAIN
VAR
(*	In USA/UK the CSV field separator is a comma.
	In Germany and some other European countries the CSV field separator is a semicolon. *)
	bChangeSeparatorToComma	: BOOL := TRUE;
	iLoopDMXCtrlQ			: INT;
	ENBufferMgmt			: ENUM_BufferMgmt;
	diMapTest				: DINT;
	arrfFnGenerVal			: ARRAY[0..gc.uiMaxNrOfDMXChannel] OF LREAL;
	uiIndexFnGenSend		: UINT;
	uiIndexFnGenRtn			: UINT;
	uiLoopDebouncePNPII		: UINT;
	uiLoopDebounceNPNII		: UINT;
END_VAR

IF bChangeSeparatorToComma THEN
	DEFAULT_CSV_FIELD_SEP := 16#2C;(* Comma ASCII code *)
ELSE
	DEFAULT_CSV_FIELD_SEP := 16#3B;(* Semicolon ASCII code *)
END_IF

P_TextModeRead();(* This sample program opens and reads CSV file in text mode *)

P_TextModeWrite();(* This sample program opens and writes CSV file in text mode *)

P_BinaryModeRead();(* This sample program opens and reads CSV file in binary mode *)

P_BinaryModeWrite();(* This sample program opens and writes CSV file in binary mode *)

P_ArgToConvExample();(* This sample program shows the usage of the ARG_TO_CSVFIELD and CSVFILED_TO_ARG conversion functions *)

P_StringToConvExample();(* This sample program shows the usage of the STRING_TO_CSVFIELD and CSVFIELD_TO_STRING conversion functions *)

//DMX Code
//Special case to handle function calls outside ("send" and "return" to FB for SIN (or potentially other) function output types)
//IF gFB.arrFB_DMX[uiIndexFnGenSend].I.ENWaveform = ENUM_I_Waveform.EN_Sin THEN
//	FOR uiIndexFnGenSend := 0 TO gc.uiMaxNrOfDMXChannel BY 1 DO
//		//SIN Function MUST be called from MAIN; not within FunctionBlock (FB_DMX)
//		arrfFnGenerVal[uiIndexFnGenSend]	:= 1+(SIN(g_ast.DMX[uiIndexFnGenSend].I.fFnGenerValTempSin));
//	END_FOR
	
//	FOR uiIndexFnGenRtn := 0 TO gc.uiMaxNrOfDMXChannel BY 1 DO
//		//SIN Function MUST be called from MAIN; not within FunctionBlock (FB_DMX)
//		gFB.arrFB_DMX[uiIndexFnGenRtn].I.fFnGenerValRtn	:= arrfFnGenerVal[uiIndexFnGenRtn];
//	END_FOR
//END_IF

//Link AST to hardware inputs - PNP
FOR uiLoopDebouncePNPII	:= 0 TO gc.uiMaxNrDMXTestCh BY 1 DO
	g_ast.arrFBIntPNP[uiLoopDebouncePNPII].IQ.xTrig		:= g_ast.arrInputPNP[uiLoopDebouncePNPII];
END_FOR

//Link AST to hardware inputs - NPN
FOR uiLoopDebounceNPNII	:= 0 TO gc.uiMaxNrDMXTestCh BY 1 DO
	g_ast.arrFBIntNPN[uiLoopDebounceNPNII].IQ.xTrig		:= g_ast.arrInputNPN[uiLoopDebounceNPNII];
END_FOR

END_PROGRAM

// ---- POUs/P_TextModeWrite.TcPOU
(* Writing of CSV file in text mode. None of the field value is containing any non-printing control characters like line feed, carriage return, quotation marks, semicolon... *)
PROGRAM P_TextModeWrite
VAR
	bWrite			: BOOL := FALSE;(* Rising edge starts program execution *)
	sNetId			: T_AmsNetId := '';	(* TwinCAT system network address *)
	sFileName		: T_MaxString; (* := 'C:\Beck\Result.csv'*) (* CSV destination file path and name *)
	sCSVLine		: T_MaxString := '';(* Single CSV text line (row, record), we are using string as record buffer (your are able to see created fields) *)
	sCSVField		: T_MaxString := '';(* Single CSV field value (column, record field) *)
	bBusy			: BOOL;
	bError			: BOOL;
	nErrId			: UDINT;
	nRow	 		: UDINT 	:= gc.uiMaxNrDMXTestCh;(* Row number (record) *)
	nColumn			: UDINT 	:= 2;(* Column number (record field) *)
	hFile			: UINT		:= 0;(* File handle of the source file *)
	step			: DWORD 	:= 0;
	fbFileOpen		: FB_FileOpen;(* Opens file *)
	fbFileClose		: FB_FileClose;(* Closes file *)
	fbFilePuts		: FB_FilePuts;(* Writes one record (line) *)
	fbWriter		: FB_CSVMemBufferWriter;(* Helper function block used to create CSV data bytes (single record line) *)

	sDUTIDNr		: STRING(255); //Device Under Test ID Number
	r_tSaveResultFile		: R_TRIG;
	r_tUpdateTimestamp		: R_TRIG;
	funcSystemTime	: NT_GetTime;
	tstSystemTime	: TIMESTRUCT;
	sYearDash		: STRING(5);
	sMonthDash		: STRING(3);
	sDayComma		: STRING(3);
	sHourColon		: STRING(3);
	sMinuteColon	: STRING(3);
	sMinSec			: STRING(5);
	sHourMinSec		: STRING(8);
	sYearMonth		: STRING(8);
	sYearMonthDay	: STRING(11);
	sTimestamp		: STRING(19);
	sFilenameUnique	: STRING(255);
	sFileDir		: STRING(255);
	sFileExtension	: STRING(10);
	sFileNameNoExtension	: STRING(255);	
	
	database		: ARRAY[0..MAX_CSV_ROWS, 0..MAX_CSV_COLUMNS ] OF STRING(MAX_CSV_FIELD_LENGTH); (*:=[ (* Source PLC database *)
	'0_0', '0_1', '0_2', '0_3', '0_4', '0_5',
	'1_0', '1_1', '1_2', '1_3', '1_4', '1_5',
	'2_0', '2_1', '2_2', '2_3', '2_4', '2_5',
	'3_0', '3_1', '3_2', '3_3', '3_4', '3_5',
	'4_0', '4_1', '4_2', '4_3', '4_4', '4_5',
	'5_0', '5_1', '5_2', '5_3', '5_4', '5_5'];*)
END_VAR

r_tSaveResultFile();
r_tUpdateTimestamp();

funcSystemTime(START:=r_tUpdateTimestamp.Q);
tstSystemTime	:= funcSystemTime.TIMESTR;
sYearDash	:= CONCAT(STR1:=WORD_TO_STRING(tstSystemTime.wYear),STR2:='-');
sMonthDash	:= CONCAT(STR1:=WORD_TO_STRING(tstSystemTime.wMonth),STR2:='-');
sDayComma	:= CONCAT(STR1:=WORD_TO_STRING(tstSystemTime.wDay),STR2:=',');
sHourColon	:= CONCAT(STR1:=WORD_TO_STRING(tstSystemTime.wHour),STR2:=':');
sMinuteColon:= CONCAT(STR1:=WORD_TO_STRING(tstSystemTime.wMinute),STR2:=':');
sMinSec		:= CONCAT(STR1:=sMinuteColon,STR2:=WORD_TO_STRING(tstSystemTime.wSecond));
sHourMinSec	:= CONCAT(STR1:=sHourColon,sMinSec);
sYearMonth	:= CONCAT(STR1:=sYearDash,STR2:=sMonthDash);
sYearMonthDay	:= CONCAT(STR1:=sYearMonth,STR2:=sDayComma);
sTimestamp	:= CONCAT(STR1:=sYearMonthDay,STR2:=sHourMinSec);
sFilenameUnique	:= CONCAT(STR1:=sTimestamp,STR2:=sDUTIDNr);
sFileNameNoExtension	:= CONCAT(STR1:=sFileDir,STR2:=sFilenameUnique);
sFileName	:= CONCAT(STR1:=sFileNameNoExtension,STR2:=sFileExtension);

CASE step OF
	0:	(* Wait for rising edge at bWrite variable *)
		IF bWrite THEN
			bWrite 	:= FALSE;
			bBusy 	:= TRUE;
			bError	:= FALSE;
			nErrId	:= 0;
			hFile	:= 0;
			nRow	:= 0;
			nColumn	:= 0;
			step 	:= 1;
		END_IF

	1:	(* Open source file *)
		fbFileOpen(  bExecute := FALSE  );
		fbFileOpen( sNetId := sNetId, sPathName := sFileName, nMode := FOPEN_MODEWRITE OR FOPEN_MODETEXT,(* Open file in TEXT mode! *)
					ePath := PATH_GENERIC, bExecute := TRUE );
		step := 2;

	2:(* Wait until open not busy *)
		fbFileOpen( bExecute := FALSE, bError => bError, nErrID => nErrID, hFile => hFile );
		IF NOT fbFileOpen.bBusy THEN
			IF NOT fbFileOpen.bError THEN
				step := 3;
			ELSE(* Error: file not found? *)
				step := 100;
			END_IF
		END_IF

	3:(* Convert one PLC record to CSV format *)
		sCSVLine := '';
		fbWriter.eCmd := eEnumCmd_First;(* Write first field value *)
		IF nRow <= MAX_CSV_ROWS THEN

			FOR nColumn := 0 TO MAX_CSV_COLUMNS BY 1 DO

				sCSVField := STRING_TO_CSVFIELD( database[ nRow, nColumn ], FALSE );(* TODO: Get field value from application *)

				(* Add new field to the record buffer *)
				fbWriter( 	pBuffer := ADR( sCSVLine ), cbBuffer := SIZEOF( sCSVLine ) - 1, putValue := sCSVField, pValue := 0, cbValue := 0,
							bCRLF := ( nColumn = MAX_CSV_COLUMNS ) );(* bCRLF == TRUE => Write CRLF after the last field value *)
				IF fbWriter.bOk THEN
					fbWriter.eCmd := eEnumCmd_Next;(* Write next field value *)
				ELSE(* Error *)
					step := 100;
					RETURN;
				END_IF

			END_FOR(* FOR nColumn := 0... *)

			(* FB_FilePuts adds allready CR (carriage return) to the written line.
			We have to replace the $R$L characters with $L character to avoid double CR. *)
			IF RIGHT( sCSVLine, 2 ) = '$R$L' THEN
				sCSVLine := REPLACE( sCSVLine, '$L', 2, LEN( sCSVLine ) - 1 );
			END_IF

			nRow := nRow + 1;(* Increment number of created records (rows) *)
			step := 4;(* Write record to the file *)

		ELSE(* All rows written => Close file *)
			step := 10;
		END_IF

	4:	(* Write single text line *)
		fbFilePuts( bExecute := FALSE );
		fbFilePuts( sNetId := sNetId, hFile := hFile, sLine := sCSVLine, bExecute := TRUE );
		step := 5;

	5:(* Wait until write not busy *)
		fbFilePuts( bExecute := FALSE, bError => bError, nErrID => nErrID );
		IF NOT fbFilePuts.bBusy THEN
			IF NOT fbFilePuts.bError THEN
				step := 3;(* Write next record *)
			ELSE(* Error *)
				step := 100;
			END_IF
		END_IF

	10:	(* Close source file *)
		fbFileClose( bExecute := FALSE );
		fbFileClose( sNetId := sNetId, hFile := hFile, bExecute := TRUE );
		step := 11;

	11:(* Wait until close not busy *)
		fbFileClose( bExecute := FALSE, bError => bError, nErrID => nErrID );
		IF ( NOT fbFileClose.bBusy ) THEN
			hFile := 0;
			step := 100;
		END_IF

	100: (* Error or ready step => cleanup *)
		IF ( hFile <> 0 ) THEN
			step := 10; (* Close the source file *)
		ELSE
			bBusy := FALSE;
			step := 0;	(* Ready *)
		END_IF

END_CASE

END_PROGRAM

// ---- POUs/SclByteDMX.TcPOU
FUNCTION SclByteDMX : BYTE
VAR_INPUT
	byUnscaled	: BYTE;
END_VAR
VAR
END_VAR

IF byUnscaled = 0 THEN
	SclByteDMX	:= 0;
ELSE
	SclByteDMX	:= 255;
END_IF

END_FUNCTION

// ---- GlobalTextList.TcGTLO
TEXTLIST GlobalTextList
  441 = '%i'
  803 = '%s'
  91 = '(Local) Filepath of\nRecipe (.csv):\n(Tap to Edit)'
  636 = 'Current\nIndex: %i'
  758 = 'Ending Index:'
  841 = 'File Date-Time:'
  675 = 'File Extension:'
  567 = 'Global Result: %s'
  886 = 'ID# of UUT\n(Unit Under Test):'
  520 = 'Invert Recipe Settings\n+ Set Config!'
  544 = 'Load Recipe File'
  742 = 'Local Filename of Last\nSaved Result File:'
  85 = 'Reset DC Test'
  472 = 'Reset Motor Test'
  191 = 'Reset Seq DMX Test'
  698 = 'Reset Test'
  724 = 'Result File Directory:'
  28 = 'Run DC Test'
  526 = 'Run Motor Test'
  199 = 'Run Seq DMX Test'
  830 = 'Run Static Test'
  429 = 'Save Result File'
  663 = 'Set all DUT Values to:'
  599 = 'Set Routing per File'
  752 = 'Starting Index:'
  149 = 'Table of Channels\nw/ Discrepancies:'
END_TEXTLIST

// ---- VISUs/Visualization.TcVIS
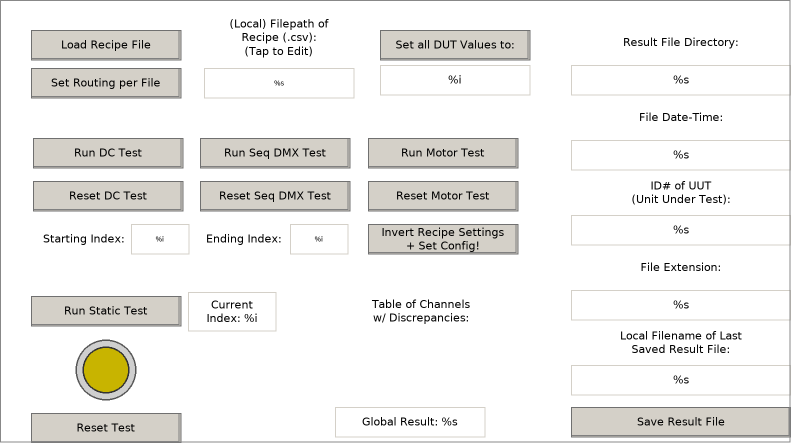
VISUALIZATION Visualization  // 791x443
    Button (31,30 150x30), "Load Recipe File", invisible if: DMXTest.iParseFile<>0
        tap P_TextModeRead.r_tFileChg.CLK
    Label (204,9 150x57), "(Local) Filepath of Recipe (.csv): (Tap to Edit)"
    Textfield (204,68 150x30), "%s", text variable: P_TextModeRead.sFilePathHMI
        OnMouseClick: write the text variable via Edit
    Textfield (335,407 150x30), "Global Result: %s"
    Label (356,296 130x30), "Table of Channels w/ Discrepancies:"
    Label (571,177 220x31), "ID# of UUT (Unit Under Test):"
    Textfield (571,215 220x30), "%s", text variable: P_TextModeWrite.sDUTIDNr
        OnMouseClick: write the text variable via VisuDialogs.Keypad
    Button (571,407 220x30), "Save Result File"
        tap P_TextModeWrite.r_tSaveResultFile.CLK
    Label (571,327 220x31), "Local Filename of Last Saved Result File:"
    Textfield (571,365 220x30), "%s", text variable: P_TextModeWrite.sFileName
    Label (571,102 220x31), "File Date-Time:"
    Textfield (571,140 220x30), "%s", text variable: P_TextModeWrite.sTimestamp
        tap P_TextModeWrite.r_tUpdateTimestamp.CLK p3779583253=TRUE
    Label (571,27 220x31), "Result File Directory:"
    Label (571,252 220x31), "File Extension:"
    Textfield (571,290 220x30), "%s", text variable: P_TextModeWrite.sFileExtension
        OnMouseClick: write the text variable via VisuDialogs.Keypad
    Textfield (571,65 220x30), "%s", text variable: P_TextModeWrite.sFileDir
        OnMouseClick: write the text variable via VisuDialogs.Keypad
    Lamp1 (71,335 70x70), variable: DMXTest.xDMXSeqTestInProgressOnce, style: Lamp-Lamp1-Yellow
    Button (31,296 150x30), "Run Static Test"
        tap DMXTest.rt_RunStaticTest.CLK
    Button (31,413 150x30), "Reset Test", invisible if: DMXTest.iCompareStaticSM<>120
        tap DMXTest.rt_ResetTest.CLK p3779583253=TRUE
    Button (31,68 150x30), "Set Routing per File", invisible if: DMXTest.iSetConfig<>0
        tap DMXTest.r_tSetConfig.CLK
    Textfield (188,292 88x39), "Current Index: %i", text variable: DMXTest.uiLoopRcvIndex
    Button (380,30 150x30), "Set all DUT Values to:"
        tap DMXTest.r_tSetDUTVal.CLK
    Textfield (380,65 150x30), "%i", text variable: DMXTest.usiDUTVal
        OnMouseClick: write the text variable via InputWithLimits, min 0, max 255
    Button (200,138 150x30), "Run Seq DMX Test"
        tap DMXTest.rt_RunSeqTestOnce.CLK p3779583253=TRUE
    Button (200,181 150x30), "Reset Seq DMX Test"
        tap DMXTest.rt_ResetTestSeq.CLK p3779583253=TRUE
    Button (33,138 150x30), "Run DC Test"
        tap DMXTest.rt_RunSeqTestOnceDC.CLK p3779583253=TRUE
    Button (33,181 150x30), "Reset DC Test"
        tap DMXTest.rt_ResetTestSeqDC.CLK p3779583253=TRUE
    Button (368,138 150x30), "Run Motor Test"
    Button (368,181 150x30), "Reset Motor Test"
    Textfield (131,224 58x30), "%i", text variable: DMXTest.uiStartingIndex
        OnMouseClick: write the text variable via Edit
    Textfield (290,224 58x30), "%i", text variable: DMXTest.uiEndingIndex
        OnMouseClick: write the text variable via Edit
    Label (44,225 80x28), "Starting Index:"
    Label (204,225 80x28), "Ending Index:"
    Button (368,224 150x30), "Invert Recipe Settings + Set Config!"
        tap DMXTest.R_TInvertRecipe.CLK p3779583253=TRUE
END_VISUALIZATION
